C05459=1024.143,54.975,397.669,167.560,48.444,158.955
C05460=1024.137,54.725,397.687,167.557,48.448,158.956
C05461=1024.131,54.476,397.703,167.554,48.453,158.956
C05462=1024.125,54.227,397.719,167.551,48.457,158.956
C05463=1024.119,53.977,397.736,167.549,48.461,158.957
C05464=1024.113,53.728,397.752,167.547,48.465,158.957
C05465=1024.107,53.479,397.769,167.544,48.469,158.958
C05466=1024.102,53.230,397.786,167.542,48.473,158.958
C05467=1024.095,52.980,397.802,167.539,48.477,158.958
C05468=1024.089,52.730,397.818,167.536,48.481,158.959
C05469=1024.083,52.481,397.835,167.534,48.485,158.959
C05470=1024.077,52.232,397.852,167.531,48.489,158.960
C05471=1024.071,51.983,397.868,167.528,48.494,158.960
C05472=1024.066,51.733,397.885,167.527,48.497,158.961
C05473=1024.060,51.484,397.901,167.524,48.501,158.961
C05474=1024.054,51.234,397.917,167.521,48.505,158.961
C05475=1024.048,50.985,397.934,167.519,48.510,158.962
C05476=1024.041,50.735,397.950,167.516,48.513,158.962
C05477=1024.035,50.486,397.967,167.513,48.517,158.962
C05478=1024.030,50.237,397.984,167.510,48.521,158.963
C05479=1024.024,49.987,398.000,167.508,48.525,158.963
C05480=1024.018,49.738,398.017,167.506,48.529,158.964
C05481=1024.012,49.489,398.033,167.503,48.533,158.964
C05482=1024.006,49.239,398.049,167.500,48.537,158.964
C05483=1024.000,48.990,398.065,167.498,48.541,158.965
C05484=1023.995,48.740,398.082,167.495,48.546,158.965
C05485=1023.989,48.491,398.098,167.493,48.549,158.966
C05486=1023.983,48.242,398.115,167.491,48.553,158.966
C05487=1023.977,47.992,398.131,167.488,48.557,158.966
C05488=1023.971,47.743,398.147,167.485,48.561,158.967
C05489=1023.965,47.494,398.164,167.483,48.566,158.967
C05490=1023.959,47.245,398.180,167.480,48.570,158.968
C05491=1023.954,46.995,398.197,167.478,48.573,158.968
C05492=1023.948,46.746,398.214,167.475,48.577,158.968
C05493=1023.942,46.496,398.230,167.472,48.581,158.969
C05494=1023.935,46.246,398.246,167.470,48.585,158.969
C05495=1023.929,45.997,398.263,167.467,48.589,158.969
C05496=1023.923,45.748,398.279,167.464,48.593,158.970
C05497=1023.917,45.498,398.295,167.463,48.597,158.970
C05498=1023.912,45.249,398.312,167.460,48.601,158.971
C05499=1023.906,44.999,398.328,167.457,48.605,158.971
C05500=1023.901,44.751,398.344,167.454,48.609,158.971
C05501=1023.895,44.501,398.360,167.452,48.613,158.972
C05502=1023.889,44.252,398.377,167.449,48.617,158.972
C05503=1023.883,44.003,398.393,167.447,48.621,158.973
C05504=1023.876,43.717,398.411,167.444,48.625,158.973
C05505=1023.870,43.433,398.430,167.441,48.630,158.973
C05506=1023.863,43.148,398.449,167.439,48.634,158.974
C05507=1023.857,42.863,398.467,167.435,48.638,158.974
C05508=1023.851,42.614,398.484,167.432,48.642,158.974
C05509=1023.845,42.364,398.499,167.431,48.647,158.975
C05510=1023.839,42.115,398.516,167.428,48.651,158.975
C05511=1023.833,41.865,398.531,167.425,48.654,158.976
C05512=1023.827,41.616,398.547,167.422,48.658,158.976
C05513=1023.821,41.366,398.564,167.420,48.663,158.977
C05514=1023.815,41.117,398.580,167.417,48.667,158.977
C05515=1023.809,40.868,398.596,167.414,48.671,158.977
C05516=1023.804,40.618,398.612,167.412,48.675,158.978
C05517=1023.797,40.369,398.627,167.409,48.679,158.978
C05518=1023.791,40.119,398.644,167.407,48.683,158.978
C05519=1023.785,39.870,398.660,167.405,48.687,158.979
C05520=1023.779,39.620,398.675,167.402,48.691,158.979
C05521=1023.773,39.371,398.692,167.399,48.695,158.980
C05522=1023.767,39.121,398.708,167.397,48.699,158.980
C05523=1023.761,38.872,398.724,167.394,48.703,158.980
C05524=1023.756,38.623,398.739,167.391,48.707,158.981
C05525=1023.750,38.374,398.755,167.388,48.711,158.981
C05526=1023.744,38.124,398.771,167.387,48.715,158.982
C05527=1023.738,37.874,398.787,167.384,48.719,158.982
C05528=1023.732,37.625,398.803,167.381,48.723,158.982
C05529=1023.726,37.376,398.819,167.378,48.727,158.983
C05530=1023.720,37.126,398.834,167.376,48.731,158.983
C05531=1023.714,36.877,398.850,167.373,48.736,158.983
C05532=1023.708,36.627,398.867,167.370,48.740,158.984
C05533=1023.702,36.377,398.882,167.368,48.744,158.984
C05534=1023.696,36.129,398.898,167.365,48.747,158.984
C05535=1023.691,35.879,398.913,167.363,48.752,158.985
C05536=1023.684,35.630,398.929,167.361,48.756,158.985
C05537=1023.678,35.380,398.944,167.358,48.760,158.986
C05538=1023.672,35.131,398.961,167.356,48.764,158.986
C05539=1023.666,34.881,398.975,167.353,48.768,158.987
C05540=1023.660,34.632,398.992,167.350,48.772,158.987
C05541=1023.654,34.382,399.007,167.348,48.777,158.987
C05542=1023.648,34.133,399.023,167.345,48.781,158.988
C05543=1023.643,33.883,399.038,167.342,48.785,158.988
C05544=1023.636,33.634,399.054,167.339,48.789,158.988
C05545=1023.630,33.384,399.069,167.337,48.793,158.989
C05546=1023.624,33.135,399.085,167.334,48.797,158.989
C05547=1023.618,32.885,399.101,167.331,48.801,158.990
C05548=1023.612,32.636,399.117,167.329,48.805,158.990
C05549=1023.606,32.387,399.131,167.327,48.809,158.991
C05550=1023.600,32.138,399.148,167.324,48.813,158.991
C05551=1023.594,31.888,399.163,167.322,48.817,158.991
C05552=1023.588,31.639,399.179,167.319,48.821,158.992
C05553=1023.582,31.389,399.194,167.316,48.826,158.992
C05554=1023.576,31.141,399.210,167.314,48.830,158.992
C05555=1023.571,30.891,399.225,167.311,48.834,158.993
C05556=1023.564,30.641,399.240,167.308,48.837,158.993
C05557=1023.558,30.392,399.256,167.305,48.841,158.993
C05558=1023.553,30.142,399.272,167.303,48.846,158.994
C05559=1023.546,29.893,399.287,167.300,48.850,158.994
C05560=1023.541,29.643,399.303,167.298,48.854,158.995
C05561=1023.534,29.394,399.318,167.296,48.858,158.995
C05562=1023.528,29.144,399.334,167.293,48.861,158.995
C05563=1023.523,28.894,399.350,167.290,48.866,158.996
C05564=1023.517,28.645,399.364,167.288,48.870,158.996
C05565=1023.511,28.396,399.380,167.285,48.874,158.996
C05566=1023.505,28.146,399.395,167.282,48.878,158.997
C05567=1023.499,27.897,399.412,167.279,48.882,158.997
C05568=1023.492,27.612,399.428,167.277,48.887,158.998
C05569=1023.485,27.327,399.445,167.273,48.891,158.998
C05570=1023.479,27.043,399.463,167.271,48.896,158.999
C05571=1023.472,26.758,399.481,167.268,48.901,158.999
C05572=1023.466,26.508,399.496,167.265,48.905,158.999
C05573=1023.460,26.259,399.512,167.262,48.909,159.000
C05574=1023.453,26.009,399.527,167.259,48.913,159.000
C05575=1023.448,25.760,399.542,167.257,48.917,159.000
C05576=1023.442,25.510,399.557,167.255,48.921,159.001
C05577=1023.435,25.261,399.573,167.252,48.925,159.001
C05578=1023.430,25.011,399.588,167.250,48.929,159.002
C05579=1023.424,24.762,399.603,167.247,48.934,159.002
C05580=1023.417,24.513,399.618,167.244,48.938,159.002
C05581=1023.412,24.263,399.633,167.242,48.942,159.003
C05582=1023.406,24.014,399.648,167.239,48.945,159.003
C05583=1023.399,23.765,399.663,167.237,48.950,159.004
C05584=1023.394,23.515,399.679,167.234,48.954,159.004
C05585=1023.388,23.266,399.694,167.231,48.958,159.004
C05586=1023.381,23.016,399.709,167.228,48.962,159.005
C05587=1023.376,22.766,399.724,167.226,48.967,159.005
C05588=1023.369,22.517,399.739,167.223,48.971,159.005
C05589=1023.364,22.268,399.754,167.220,48.974,159.006
C05590=1023.358,22.018,399.769,167.218,48.978,159.006
C05591=1023.352,21.768,399.784,167.215,48.982,159.006
C05592=1023.346,21.520,399.799,167.212,48.987,159.007
C05593=1023.340,21.270,399.815,167.210,48.991,159.007
C05594=1023.334,21.020,399.830,167.207,48.995,159.008
C05595=1023.328,20.771,399.844,167.205,48.999,159.008
C05596=1023.322,20.521,399.860,167.202,49.003,159.008
C05597=1023.316,20.272,399.875,167.200,49.006,159.009
C05598=1023.310,20.023,399.890,167.197,49.011,159.009
C05599=1023.304,19.773,399.905,167.194,49.015,159.009
C05600=1023.299,19.524,399.920,167.192,49.019,159.010
C05601=1023.292,19.274,399.935,167.189,49.023,159.010
C05602=1023.286,19.024,399.950,167.186,49.027,159.010
C05603=1023.281,18.775,399.965,167.184,49.032,159.011
C05604=1023.274,18.525,399.980,167.181,49.036,159.011
C05605=1023.268,18.276,399.995,167.178,49.039,159.012
C05606=1023.262,18.027,400.009,167.175,49.043,159.012
C05607=1023.257,17.777,400.025,167.173,49.047,159.012
C05608=1023.251,17.528,400.039,167.170,49.052,159.013
C05609=1023.245,17.278,400.054,167.168,49.056,159.013
C05610=1023.238,17.028,400.068,167.165,49.060,159.013
C05611=1023.232,16.779,400.083,167.162,49.064,159.014
C05612=1023.226,16.529,400.098,167.160,49.069,159.014
C05613=1023.221,16.280,400.113,167.157,49.073,159.015
C05614=1023.215,16.030,400.128,167.154,49.077,159.015
C05615=1023.209,15.781,400.143,167.151,49.080,159.015
C05616=1023.203,15.532,400.158,167.149,49.084,159.015
C05617=1023.196,15.282,400.173,167.146,49.088,159.016
C05618=1023.191,15.032,400.187,167.144,49.093,159.016
C05619=1023.185,14.783,400.202,167.142,49.097,159.017
C05620=1023.179,14.534,400.217,167.139,49.101,159.017
C05621=1023.173,14.284,400.232,167.136,49.105,159.017
C05622=1023.167,14.035,400.246,167.134,49.109,159.018
C05623=1023.161,13.785,400.261,167.131,49.113,159.018
C05624=1023.156,13.535,400.276,167.128,49.117,159.018
C05625=1023.150,13.286,400.290,167.126,49.121,159.019
C05626=1023.142,13.036,400.305,167.123,49.125,159.019
C05627=1023.137,12.787,400.319,167.120,49.129,159.020
C05628=1023.131,12.537,400.334,167.118,49.134,159.020
C05629=1023.125,12.288,400.348,167.115,49.138,159.020
C05630=1023.119,12.038,400.362,167.112,49.142,159.021
C05631=1023.113,11.789,400.377,167.109,49.147,159.021
C05632=1023.106,11.506,400.393,167.106,49.151,159.021
C05633=1023.099,11.222,400.410,167.103,49.156,159.022
C05634=1023.092,10.939,400.426,167.100,49.160,159.022
C05635=1023.085,10.656,400.442,167.097,49.165,159.023
C05636=1023.079,10.406,400.457,167.094,49.169,159.023
C05637=1023.073,10.157,400.472,167.092,49.174,159.024
C05638=1023.067,9.907,400.486,167.089,49.178,159.024
C05639=1023.061,9.658,400.500,167.086,49.182,159.024
C05640=1023.055,9.408,400.515,167.083,49.186,159.024
C05641=1023.049,9.159,400.529,167.081,49.190,159.025
C05642=1023.043,8.909,400.544,167.078,49.194,159.025
C05643=1023.037,8.660,400.558,167.076,49.198,159.026
C05644=1023.030,8.410,400.572,167.073,49.202,159.026
C05645=1023.025,8.161,400.586,167.070,49.207,159.026
C05646=1023.018,7.911,400.601,167.068,49.211,159.027
C05647=1023.013,7.662,400.616,167.065,49.215,159.027
C05648=1023.007,7.412,400.630,167.062,49.219,159.027
C05649=1023.001,7.163,400.645,167.059,49.223,159.028
C05650=1022.995,6.913,400.659,167.057,49.228,159.028
C05651=1022.989,6.664,400.673,167.054,49.232,159.029
C05652=1022.984,6.414,400.687,167.052,49.236,159.029
C05653=1022.976,6.165,400.702,167.049,49.240,159.029
C05654=1022.971,5.915,400.715,167.046,49.244,159.030
C05655=1022.965,5.665,400.730,167.044,49.248,159.030
C05656=1022.959,5.416,400.744,167.041,49.252,159.030
C05657=1022.953,5.167,400.759,167.038,49.256,159.031
C05658=1022.947,4.917,400.773,167.035,49.260,159.031
C05659=1022.941,4.668,400.788,167.033,49.264,159.031
C05660=1022.935,4.417,400.802,167.030,49.268,159.032
C05661=1022.929,4.169,400.816,167.027,49.272,159.032
C05662=1022.923,3.919,400.830,167.025,49.277,159.032
C05663=1022.917,3.669,400.844,167.022,49.281,159.033
C05664=1022.911,3.420,400.859,167.019,49.285,159.033
C05665=1022.905,3.170,400.873,167.017,49.289,159.033
C05666=1022.900,2.921,400.887,167.014,49.293,159.034
C05667=1022.894,2.671,400.901,167.011,49.297,159.034
C05668=1022.887,2.421,400.915,167.008,49.301,159.034
C05669=1022.882,2.172,400.929,167.006,49.305,159.035
C05670=1022.876,1.923,400.943,167.003,49.309,159.035
C05671=1022.870,1.673,400.958,167.001,49.313,159.035
C05672=1022.864,1.423,400.972,166.998,49.317,159.036
C05673=1022.859,1.174,400.986,166.995,49.321,159.036
C05674=1022.852,0.924,401.001,166.992,49.325,159.036
C05675=1022.846,0.675,401.014,166.990,49.329,159.037
C05676=1022.841,0.425,401.028,166.987,49.333,159.037
C05677=1022.834,0.176,401.043,166.984,49.337,159.037
C05678=1022.829,-0.074,401.057,166.981,49.341,159.038
C05679=1022.823,-0.324,401.071,166.979,49.345,159.038
C05680=1022.818,-0.572,401.085,166.976,49.349,159.038
C05681=1022.811,-0.823,401.100,166.973,49.353,159.039
C05682=1022.805,-1.072,401.113,166.970,49.357,159.039
C05683=1022.799,-1.321,401.127,166.968,49.361,159.039
C05684=1022.793,-1.571,401.142,166.965,49.365,159.040
C05685=1022.788,-1.821,401.155,166.962,49.369,159.040
C05686=1022.782,-2.070,401.170,166.960,49.373,159.040
C05687=1022.777,-2.319,401.184,166.957,49.377,159.041
C05688=1022.771,-2.570,401.198,166.954,49.381,159.041
C05689=1022.764,-2.819,401.211,166.951,49.385,159.041
C05690=1022.759,-3.068,401.226,166.949,49.389,159.042
C05691=1022.753,-3.317,401.240,166.946,49.393,159.042
C05692=1022.747,-3.568,401.254,166.943,49.397,159.042
C05693=1022.742,-3.817,401.268,166.940,49.401,159.042
C05694=1022.736,-4.067,401.282,166.938,49.405,159.043
C05695=1022.730,-4.315,401.296,166.935,49.410,159.043
C05696=1022.722,-4.598,401.311,166.932,49.414,159.043
C05697=1022.715,-4.879,401.327,166.928,49.419,159.044
C05698=1022.709,-5.161,401.342,166.926,49.424,159.044
C05699=1022.702,-5.442,401.358,166.922,49.429,159.045
C05700=1022.696,-5.691,401.372,166.920,49.433,159.045
C05701=1022.690,-5.941,401.385,166.917,49.437,159.045
C05702=1022.685,-6.190,401.399,166.914,49.441,159.046
C05703=1022.678,-6.440,401.412,166.911,49.445,159.046
C05704=1022.672,-6.690,401.426,166.909,49.449,159.047
C05705=1022.666,-6.939,401.439,166.906,49.453,159.047
C05706=1022.661,-7.189,401.453,166.904,49.457,159.047
C05707=1022.655,-7.438,401.467,166.900,49.462,159.047
C05708=1022.648,-7.688,401.481,166.897,49.466,159.048
C05709=1022.642,-7.937,401.494,166.894,49.470,159.048
C05710=1022.637,-8.187,401.508,166.892,49.474,159.048
C05711=1022.631,-8.436,401.521,166.889,49.478,159.049
C05712=1022.625,-8.686,401.535,166.887,49.482,159.049
C05713=1022.619,-8.935,401.548,166.884,49.486,159.049
C05714=1022.613,-9.185,401.563,166.881,49.490,159.050
C05715=1022.607,-9.435,401.576,166.878,49.495,159.050
C05716=1022.601,-9.685,401.589,166.876,49.499,159.050
C05717=1022.595,-9.934,401.602,166.873,49.503,159.051
C05718=1022.590,-10.184,401.616,166.871,49.507,159.051
C05719=1022.583,-10.433,401.629,166.867,49.512,159.051
C05720=1022.577,-10.682,401.643,166.864,49.516,159.052
C05721=1022.571,-10.933,401.657,166.861,49.520,159.052
C05722=1022.565,-11.182,401.670,166.859,49.524,159.052
C05723=1022.559,-11.431,401.684,166.856,49.528,159.053
C05724=1022.553,-11.681,401.697,166.853,49.532,159.053
C05725=1022.548,-11.930,401.711,166.851,49.536,159.053
C05726=1022.542,-12.180,401.724,166.848,49.540,159.054
C05727=1022.536,-12.430,401.738,166.845,49.544,159.054
C05728=1022.530,-12.679,401.751,166.842,49.548,159.054
C05729=1022.525,-12.928,401.765,166.840,49.552,159.054
C05730=1022.518,-13.178,401.778,166.837,49.556,159.055
C05731=1022.512,-13.428,401.792,166.835,49.560,159.055
C05732=1022.507,-13.678,401.805,166.832,49.564,159.056
C05733=1022.501,-13.928,401.819,166.828,49.569,159.056
C05734=1022.495,-14.177,401.832,166.825,49.573,159.056
C05735=1022.489,-14.426,401.845,166.823,49.577,159.056
C05736=1022.483,-14.676,401.859,166.820,49.581,159.057
C05737=1022.477,-14.925,401.872,166.817,49.585,159.057
C05738=1022.472,-15.175,401.885,166.814,49.589,159.057
C05739=1022.466,-15.424,401.899,166.812,49.593,159.058
C05740=1022.460,-15.674,401.913,166.809,49.597,159.058
C05741=1022.454,-15.924,401.925,166.806,49.601,159.058
C05742=1022.448,-16.173,401.938,166.804,49.605,159.059
C05743=1022.442,-16.422,401.952,166.801,49.609,159.059
C05744=1022.437,-16.673,401.965,166.797,49.613,159.059
C05745=1022.430,-16.922,401.978,166.795,49.618,159.060
C05746=1022.424,-17.172,401.991,166.792,49.622,159.060
C05747=1022.418,-17.421,402.004,166.789,49.626,159.060
C05748=1022.412,-17.670,402.017,166.787,49.630,159.061
C05749=1022.407,-17.920,402.030,166.784,49.634,159.061
C05750=1022.401,-18.170,402.044,166.781,49.638,159.061
C05751=1022.395,-18.420,402.056,166.777,49.642,159.061
C05752=1022.389,-18.669,402.069,166.775,49.647,159.062
C05753=1022.383,-18.919,402.082,166.772,49.651,159.062
C05754=1022.377,-19.168,402.096,166.770,49.655,159.062
C05755=1022.371,-19.417,402.109,166.767,49.659,159.063
C05756=1022.365,-19.667,402.122,166.764,49.663,159.063
C05757=1022.359,-19.917,402.135,166.762,49.667,159.063
C05758=1022.353,-20.167,402.148,166.758,49.671,159.064
C05759=1022.347,-20.416,402.161,166.755,49.675,159.064
C05760=1022.340,-20.696,402.176,166.753,49.680,159.064
C05761=1022.334,-20.976,402.191,166.749,49.685,159.065
C05762=1022.327,-21.255,402.205,166.746,49.690,159.065
C05763=1022.320,-21.535,402.220,166.743,49.694,159.065
C05764=1022.314,-21.785,402.232,166.740,49.698,159.066
C05765=1022.309,-22.035,402.245,166.738,49.702,159.066
C05766=1022.302,-22.284,402.258,166.734,49.707,159.066
C05767=1022.297,-22.533,402.270,166.731,49.711,159.067
C05768=1022.292,-22.783,402.284,166.729,49.715,159.067
C05769=1022.286,-23.033,402.297,166.726,49.719,159.067
C05770=1022.279,-23.282,402.310,166.723,49.723,159.067
C05771=1022.274,-23.532,402.323,166.720,49.727,159.068
C05772=1022.267,-23.781,402.336,166.718,49.731,159.068
C05773=1022.261,-24.031,402.348,166.715,49.735,159.068
C05774=1022.256,-24.281,402.362,166.711,49.739,159.069
C05775=1022.250,-24.530,402.375,166.709,49.743,159.069
C05776=1022.244,-24.780,402.387,166.706,49.747,159.069
C05777=1022.238,-25.029,402.400,166.703,49.751,159.069
C05778=1022.233,-25.279,402.413,166.700,49.755,159.070
C05779=1022.227,-25.529,402.425,166.698,49.759,159.070
C05780=1022.221,-25.778,402.439,166.695,49.763,159.070
C05781=1022.215,-26.028,402.452,166.692,49.767,159.071
C05782=1022.209,-26.278,402.464,166.689,49.772,159.071
C05783=1022.204,-26.527,402.477,166.686,49.776,159.071
C05784=1022.198,-26.776,402.490,166.683,49.780,159.072
C05785=1022.192,-27.026,402.502,166.681,49.784,159.072
C05786=1022.186,-27.276,402.516,166.678,49.788,159.072
C05787=1022.181,-27.526,402.529,166.675,49.792,159.072
C05788=1022.175,-27.776,402.541,166.672,49.796,159.073
C05789=1022.168,-28.025,402.553,166.669,49.800,159.073
C05790=1022.163,-28.274,402.565,166.666,49.804,159.073
C05791=1022.156,-28.524,402.579,166.664,49.809,159.074
C05792=1022.151,-28.774,402.591,166.661,49.813,159.074
C05793=1022.145,-29.023,402.604,166.658,49.817,159.074
C05794=1022.139,-29.273,402.616,166.654,49.822,159.074
C05795=1022.133,-29.523,402.629,166.652,49.826,159.075
C05796=1022.128,-29.772,402.641,166.649,49.830,159.075
C05797=1022.122,-30.022,402.654,166.646,49.834,159.075
C05798=1022.115,-30.271,402.666,166.644,49.838,159.076
C05799=1022.109,-30.521,402.679,166.641,49.842,159.076
C05800=1022.103,-30.770,402.691,166.638,49.847,159.076
C05801=1022.098,-31.020,402.704,166.635,49.851,159.077
C05802=1022.092,-31.270,402.716,166.632,49.855,159.077
C05803=1022.086,-31.520,402.729,166.629,49.859,159.077
C05804=1022.080,-31.770,402.741,166.627,49.863,159.078
C05805=1022.075,-32.019,402.754,166.623,49.867,159.078
C05806=1022.068,-32.269,402.765,166.620,49.871,159.078
C05807=1022.062,-32.518,402.778,166.618,49.875,159.078
C05808=1022.057,-32.768,402.790,166.615,49.880,159.079
C05809=1022.051,-33.018,402.803,166.612,49.884,159.079
C05810=1022.045,-33.267,402.816,166.608,49.888,159.079
C05811=1022.039,-33.517,402.829,166.606,49.892,159.079
C05812=1022.033,-33.766,402.841,166.603,49.896,159.080
C05813=1022.027,-34.015,402.853,166.600,49.900,159.080
C05814=1022.021,-34.265,402.865,166.598,49.904,159.080
C05815=1022.015,-34.514,402.877,166.594,49.908,159.081
C05816=1022.010,-34.764,402.890,166.591,49.913,159.081
C05817=1022.004,-35.014,402.903,166.589,49.917,159.081
C05818=1021.998,-35.263,402.915,166.586,49.921,159.081
C05819=1021.992,-35.513,402.927,166.583,49.925,159.082
C05820=1021.986,-35.764,402.939,166.580,49.929,159.082
C05821=1021.981,-36.013,402.951,166.577,49.933,159.082
C05822=1021.975,-36.263,402.963,166.574,49.937,159.083
C05823=1021.969,-36.512,402.976,166.571,49.941,159.083
C05824=1021.962,-36.791,402.989,166.568,49.946,159.083
C05825=1021.956,-37.070,403.004,166.565,49.950,159.084
C05826=1021.949,-37.349,403.017,166.562,49.955,159.084
C05827=1021.943,-37.627,403.031,166.558,49.960,159.084
C05828=1021.938,-37.878,403.043,166.555,49.964,159.084
C05829=1021.932,-38.127,403.055,166.553,49.968,159.085
C05830=1021.926,-38.376,403.067,166.550,49.972,159.085
C05831=1021.920,-38.626,403.080,166.547,49.976,159.085
C05832=1021.915,-38.876,403.092,166.545,49.980,159.086
C05833=1021.909,-39.125,403.105,166.541,49.984,159.086
C05834=1021.903,-39.375,403.117,166.538,49.988,159.086
C05835=1021.897,-39.625,403.128,166.536,49.993,159.086
C05836=1021.891,-39.875,403.141,166.533,49.997,159.087
C05837=1021.885,-40.124,403.152,166.529,50.001,159.087
C05838=1021.880,-40.374,403.164,166.526,50.005,159.087
C05839=1021.873,-40.624,403.176,166.524,50.009,159.087
C05840=1021.868,-40.873,403.188,166.521,50.013,159.088
C05841=1021.862,-41.123,403.201,166.517,50.018,159.088
C05842=1021.856,-41.372,403.212,166.515,50.022,159.088
C05843=1021.850,-41.622,403.224,166.512,50.026,159.089
C05844=1021.844,-41.871,403.236,166.510,50.030,159.089
C05845=1021.838,-42.121,403.247,166.506,50.035,159.089
C05846=1021.832,-42.371,403.260,166.503,50.039,159.089
C05847=1021.826,-42.620,403.272,166.501,50.043,159.090
C05848=1021.821,-42.871,403.283,166.498,50.047,159.090
C05849=1021.815,-43.120,403.295,166.494,50.051,159.090
C05850=1021.809,-43.369,403.308,166.491,50.055,159.091
C05851=1021.803,-43.619,403.319,166.489,50.059,159.091
C05852=1021.797,-43.869,403.331,166.486,50.064,159.091
C05853=1021.792,-44.119,403.343,166.483,50.068,159.091
C05854=1021.786,-44.368,403.354,166.480,50.072,159.092
C05855=1021.780,-44.617,403.367,166.477,50.076,159.092
C05856=1021.774,-44.868,403.378,166.474,50.080,159.092
C05857=1021.769,-45.117,403.390,166.472,50.084,159.092
C05858=1021.762,-45.367,403.401,166.468,50.089,159.093
C05859=1021.757,-45.616,403.414,166.465,50.093,159.093
C05860=1021.751,-45.866,403.425,166.462,50.097,159.093
C05861=1021.745,-46.115,403.437,166.460,50.101,159.094
C05862=1021.740,-46.366,403.449,166.456,50.105,159.094
C05863=1021.734,-46.615,403.460,166.453,50.109,159.094
C05864=1021.728,-46.865,403.473,166.451,50.113,159.094
C05865=1021.722,-47.114,403.484,166.448,50.117,159.095
C05866=1021.717,-47.363,403.496,166.445,50.121,159.095
C05867=1021.710,-47.614,403.507,166.442,50.126,159.095
C05868=1021.705,-47.863,403.519,166.439,50.130,159.095
C05869=1021.699,-48.113,403.531,166.436,50.134,159.096
C05870=1021.693,-48.362,403.543,166.434,50.138,159.096
C05871=1021.688,-48.613,403.555,166.430,50.142,159.096
C05872=1021.682,-48.862,403.566,166.427,50.147,159.096
C05873=1021.677,-49.111,403.578,166.424,50.150,159.097
C05874=1021.670,-49.362,403.589,166.421,50.154,159.097
C05875=1021.665,-49.611,403.601,166.419,50.158,159.097
C05876=1021.659,-49.861,403.612,166.415,50.162,159.097
C05877=1021.653,-50.110,403.625,166.412,50.167,159.098
C05878=1021.648,-50.360,403.636,166.410,50.171,159.098
C05879=1021.642,-50.610,403.647,166.407,50.175,159.098
C05880=1021.636,-50.859,403.659,166.403,50.179,159.098
C05881=1021.631,-51.109,403.670,166.401,50.183,159.099
C05882=1021.625,-51.359,403.682,166.398,50.187,159.099
C05883=1021.619,-51.608,403.693,166.394,50.192,159.099
C05884=1021.612,-51.858,403.705,166.392,50.196,159.099
C05885=1021.607,-52.107,403.715,166.389,50.201,159.100
C05886=1021.602,-52.357,403.727,166.385,50.205,159.100
C05887=1021.595,-52.607,403.738,166.383,50.209,159.100
C05888=1021.589,-52.855,403.749,166.380,50.213,159.101
C05889=1021.583,-53.103,403.761,166.376,50.217,159.101
C05890=1021.578,-53.350,403.771,166.374,50.222,159.101
C05891=1021.572,-53.597,403.783,166.371,50.226,159.101
C05892=1021.566,-53.845,403.794,166.368,50.231,159.102
C05893=1021.560,-54.093,403.805,166.365,50.235,159.102
C05894=1021.554,-54.341,403.815,166.362,50.239,159.102
C05895=1021.548,-54.589,403.827,166.360,50.243,159.103
C05896=1021.543,-54.838,403.838,166.356,50.247,159.103
C05897=1021.537,-55.088,403.849,166.353,50.251,159.103
C05898=1021.531,-55.338,403.860,166.351,50.256,159.103
C05899=1021.525,-55.587,403.871,166.347,50.260,159.103
C05900=1021.520,-55.837,403.883,166.344,50.264,159.104
C05901=1021.514,-56.087,403.894,166.342,50.268,159.104
C05902=1021.508,-56.337,403.905,166.338,50.273,159.104
C05903=1021.502,-56.586,403.916,166.335,50.277,159.105
C05904=1021.496,-56.835,403.927,166.333,50.281,159.105
C05905=1021.490,-57.085,403.938,166.329,50.286,159.105
C05906=1021.484,-57.335,403.949,166.326,50.290,159.105
C05907=1021.478,-57.584,403.960,166.324,50.294,159.106
C05908=1021.472,-57.868,403.973,166.320,50.299,159.106
C05909=1021.465,-58.151,403.985,166.317,50.304,159.106
C05910=1021.459,-58.434,403.998,166.313,50.309,159.107
C05911=1021.452,-58.717,404.010,166.310,50.313,159.107
C05912=1021.447,-58.968,404.022,166.307,50.317,159.107
C05913=1021.441,-59.217,404.033,166.303,50.322,159.107
C05914=1021.435,-59.467,404.044,166.301,50.326,159.108
C05915=1021.429,-59.716,404.055,166.298,50.330,159.108
C05916=1021.424,-59.966,404.065,166.294,50.334,159.108
C05917=1021.417,-60.216,404.077,166.292,50.338,159.108
C05918=1021.411,-60.465,404.088,166.289,50.342,159.109
C05919=1021.406,-60.715,404.098,166.285,50.347,159.109
C05920=1021.401,-60.964,404.110,166.283,50.352,159.109
C05921=1021.395,-61.214,404.121,166.280,50.356,159.110
C05922=1021.389,-61.463,404.132,166.277,50.359,159.110
C05923=1021.383,-61.714,404.142,166.273,50.363,159.110
C05924=1021.377,-61.964,404.153,166.271,50.368,159.110
C05925=1021.372,-62.213,404.164,166.268,50.372,159.110
C05926=1021.366,-62.463,404.175,166.264,50.376,159.111
C05927=1021.360,-62.712,404.186,166.262,50.380,159.111
C05928=1021.355,-62.962,404.197,166.259,50.384,159.111
C05929=1021.350,-63.212,404.208,166.255,50.389,159.111
C05930=1021.343,-63.462,404.219,166.253,50.393,159.112
C05931=1021.338,-63.712,404.229,166.250,50.397,159.112
C05932=1021.332,-63.961,404.240,166.246,50.401,159.112
C05933=1021.326,-64.211,404.251,166.244,50.405,159.112
C05934=1021.321,-64.460,404.262,166.241,50.410,159.113
C05935=1021.315,-64.710,404.273,166.238,50.414,159.113
C05936=1021.309,-64.959,404.284,166.235,50.418,159.113
C05937=1021.304,-65.209,404.294,166.232,50.422,159.113
C05938=1021.298,-65.459,404.305,166.229,50.426,159.114
C05939=1021.293,-65.709,404.316,166.226,50.431,159.114
C05940=1021.287,-65.958,404.327,166.223,50.435,159.114
C05941=1021.282,-66.208,404.337,166.220,50.438,159.114
C05942=1021.276,-66.458,404.348,166.217,50.442,159.114
C05943=1021.270,-66.708,404.360,166.213,50.447,159.115
C05944=1021.264,-66.957,404.370,166.211,50.451,159.115
C05945=1021.258,-67.208,404.381,166.208,50.455,159.115
C05946=1021.253,-67.457,404.391,166.204,50.459,159.115
C05947=1021.247,-67.707,404.402,166.202,50.463,159.116
C05948=1021.241,-67.956,404.413,166.199,50.468,159.116
C05949=1021.236,-68.206,404.423,166.196,50.472,159.116
C05950=1021.230,-68.456,404.434,166.192,50.475,159.116
C05951=1021.225,-68.705,404.446,166.190,50.480,159.116
C05952=1021.219,-68.986,404.457,166.186,50.485,159.117
C05953=1021.213,-69.266,404.469,166.184,50.489,159.117
C05954=1021.207,-69.547,404.481,166.180,50.493,159.117
C05955=1021.201,-69.826,404.493,166.177,50.498,159.117
C05956=1021.195,-70.076,404.504,166.174,50.502,159.118
C05957=1021.189,-70.326,404.514,166.170,50.506,159.118
C05958=1021.184,-70.576,404.525,166.167,50.510,159.118
C05959=1021.178,-70.825,404.536,166.165,50.514,159.118
C05960=1021.172,-71.075,404.546,166.162,50.519,159.119
C05961=1021.167,-71.325,404.557,166.158,50.522,159.119
C05962=1021.161,-71.575,404.567,166.155,50.526,159.119
C05963=1021.156,-71.824,404.578,166.153,50.530,159.119
C05964=1021.150,-72.074,404.589,166.150,50.535,159.119
C05965=1021.144,-72.324,404.599,166.146,50.539,159.120
C05966=1021.139,-72.573,404.610,166.143,50.542,159.120
C05967=1021.133,-72.823,404.620,166.140,50.547,159.120
C05968=1021.129,-73.073,404.631,166.138,50.551,159.120
C05969=1021.123,-73.323,404.641,166.134,50.555,159.120
C05970=1021.118,-73.572,404.652,166.131,50.559,159.121
C05971=1021.112,-73.822,404.662,166.128,50.563,159.121
C05972=1021.106,-74.072,404.673,166.126,50.567,159.121
C05973=1021.101,-74.322,404.683,166.122,50.571,159.121
C05974=1021.095,-74.571,404.694,166.119,50.575,159.121
C05975=1021.090,-74.821,404.704,166.117,50.579,159.122
C05976=1021.083,-75.071,404.715,166.113,50.584,159.122
C05977=1021.079,-75.320,404.724,166.110,50.588,159.122
C05978=1021.073,-75.570,404.735,166.108,50.592,159.122
C05979=1021.067,-75.820,404.746,166.104,50.597,159.123
C05980=1021.061,-76.069,404.755,166.101,50.601,159.123
C05981=1021.056,-76.320,404.765,166.098,50.604,159.123
C05982=1021.050,-76.569,404.776,166.095,50.609,159.123
C05983=1021.045,-76.819,404.786,166.092,50.613,159.123
C05984=1021.039,-77.068,404.795,166.089,50.617,159.124
C05985=1021.033,-77.318,404.806,166.086,50.621,159.124
C05986=1021.028,-77.568,404.817,166.083,50.625,159.124
C05987=1021.022,-77.818,404.827,166.080,50.629,159.124
C05988=1021.016,-78.068,404.836,166.077,50.634,159.124
C05989=1021.011,-78.317,404.847,166.074,50.638,159.125
C05990=1021.006,-78.567,404.857,166.071,50.642,159.125
C05991=1021.000,-78.817,404.867,166.068,50.647,159.125
C05992=1020.994,-79.067,404.877,166.065,50.651,159.125
C05993=1020.988,-79.316,404.888,166.062,50.654,159.126
C05994=1020.983,-79.565,404.897,166.058,50.659,159.126
C05995=1020.978,-79.816,404.907,166.056,50.663,159.126
C05996=1020.972,-80.065,404.917,166.053,50.667,159.126
C05997=1020.966,-80.315,404.927,166.049,50.671,159.126
C05998=1020.962,-80.565,404.937,166.047,50.675,159.127
C05999=1020.955,-80.814,404.947,166.043,50.680,159.127
C06000=1020.950,-81.064,404.957,166.040,50.684,159.127
C06001=1020.944,-81.314,404.967,166.038,50.688,159.127
C06002=1020.939,-81.563,404.977,166.034,50.693,159.128
C06003=1020.933,-81.813,404.986,166.031,50.697,159.128
C06004=1020.927,-82.063,404.997,166.028,50.702,159.128
C06005=1020.921,-82.313,405.006,166.025,50.706,159.128
C06006=1020.915,-82.562,405.015,166.023,50.710,159.129
C06007=1020.910,-82.812,405.025,166.019,50.715,159.129
C06008=1020.904,-83.062,405.035,166.016,50.719,159.129
C06009=1020.898,-83.312,405.045,166.013,50.723,159.129
C06010=1020.893,-83.561,405.054,166.010,50.727,159.130
C06011=1020.887,-83.811,405.065,166.007,50.732,159.130
C06012=1020.881,-84.061,405.074,166.004,50.736,159.130
C06013=1020.876,-84.311,405.084,166.001,50.740,159.130
C06014=1020.870,-84.560,405.094,165.997,50.745,159.130
C06015=1020.865,-84.811,405.104,165.995,50.749,159.131
C06016=1020.859,-85.093,405.114,165.991,50.753,159.131
C06017=1020.852,-85.375,405.125,165.988,50.758,159.131
C06018=1020.846,-85.657,405.137,165.984,50.763,159.131
C06019=1020.840,-85.940,405.147,165.981,50.768,159.132
C06020=1020.834,-86.189,405.156,165.978,50.772,159.132
C06021=1020.829,-86.439,405.167,165.974,50.777,159.132
C06022=1020.822,-86.689,405.176,165.972,50.781,159.132
C06023=1020.818,-86.939,405.186,165.969,50.785,159.133
C06024=1020.811,-87.188,405.195,165.965,50.789,159.133
C06025=1020.806,-87.439,405.204,165.963,50.794,159.133
C06026=1020.801,-87.688,405.214,165.959,50.798,159.133
C06027=1020.795,-87.938,405.224,165.956,50.802,159.133
C06028=1020.790,-88.187,405.233,165.953,50.806,159.133
C06029=1020.784,-88.437,405.243,165.950,50.810,159.134
C06030=1020.778,-88.687,405.253,165.947,50.814,159.134
C06031=1020.773,-88.936,405.262,165.944,50.818,159.134
C06032=1020.767,-89.187,405.272,165.941,50.823,159.134
C06033=1020.762,-89.436,405.281,165.938,50.827,159.135
C06034=1020.756,-89.686,405.291,165.935,50.831,159.135
C06035=1020.751,-89.935,405.300,165.932,50.836,159.135
C06036=1020.745,-90.185,405.310,165.929,50.840,159.135
C06037=1020.740,-90.435,405.319,165.925,50.844,159.135
C06038=1020.734,-90.685,405.329,165.923,50.848,159.136
C06039=1020.729,-90.934,405.338,165.920,50.852,159.136
C06040=1020.723,-91.184,405.348,165.916,50.856,159.136
C06041=1020.718,-91.434,405.357,165.913,50.860,159.136
C06042=1020.712,-91.684,405.367,165.911,50.865,159.136
C06043=1020.707,-91.933,405.376,165.907,50.869,159.137
C06044=1020.702,-92.184,405.385,165.904,50.873,159.137
C06045=1020.696,-92.433,405.394,165.902,50.877,159.137
C06046=1020.691,-92.683,405.405,165.898,50.882,159.137
C06047=1020.685,-92.932,405.414,165.895,50.886,159.138
C06048=1020.680,-93.183,405.423,165.892,50.889,159.138
C06049=1020.674,-93.432,405.432,165.889,50.894,159.138
C06050=1020.669,-93.682,405.443,165.886,50.898,159.138
C06051=1020.664,-93.932,405.451,165.883,50.902,159.138
C06052=1020.657,-94.182,405.461,165.880,50.907,159.138
C06053=1020.653,-94.431,405.470,165.877,50.911,159.139
C06054=1020.647,-94.681,405.479,165.874,50.914,159.139
C06055=1020.642,-94.931,405.489,165.870,50.919,159.139
C06056=1020.637,-95.181,405.498,165.868,50.923,159.139
C06057=1020.631,-95.431,405.508,165.865,50.927,159.139
C06058=1020.626,-95.680,405.517,165.861,50.932,159.140
C06059=1020.620,-95.930,405.526,165.858,50.935,159.140
C06060=1020.615,-96.180,405.536,165.856,50.939,159.140
C06061=1020.609,-96.430,405.544,165.852,50.944,159.140
C06062=1020.604,-96.679,405.554,165.849,50.948,159.140
C06063=1020.599,-96.929,405.563,165.847,50.952,159.141
C06064=1020.593,-97.179,405.572,165.843,50.956,159.140
C06065=1020.588,-97.428,405.582,165.840,50.960,159.141
C06066=1020.582,-97.679,405.591,165.838,50.964,159.141
C06067=1020.577,-97.928,405.601,165.834,50.969,159.141
C06068=1020.572,-98.178,405.609,165.831,50.973,159.141
C06069=1020.566,-98.428,405.618,165.829,50.977,159.142
C06070=1020.561,-98.677,405.627,165.825,50.981,159.142
C06071=1020.555,-98.927,405.636,165.822,50.986,159.142
C06072=1020.549,-99.177,405.645,165.819,50.990,159.142
C06073=1020.545,-99.427,405.654,165.816,50.994,159.142
C06074=1020.539,-99.677,405.663,165.813,50.998,159.143
C06075=1020.533,-99.926,405.672,165.810,51.003,159.143
C06076=1020.528,-100.176,405.681,165.807,51.007,159.143
C06077=1020.523,-100.426,405.689,165.803,51.011,159.143
C06078=1020.516,-100.676,405.699,165.800,51.015,159.143
C06079=1020.511,-100.925,405.708,165.798,51.019,159.144
C06080=1020.505,-101.210,405.718,165.794,51.024,159.144
C06081=1020.499,-101.495,405.728,165.791,51.029,159.144
C06082=1020.493,-101.779,405.738,165.787,51.034,159.144
C06083=1020.486,-102.063,405.748,165.784,51.039,159.145
C06084=1020.482,-102.313,405.757,165.780,51.043,159.145
C06085=1020.476,-102.563,405.766,165.777,51.047,159.145
C06086=1020.470,-102.814,405.775,165.775,51.051,159.145
C06087=1020.465,-103.063,405.784,165.771,51.056,159.145
C06088=1020.460,-103.312,405.793,165.768,51.060,159.146
C06089=1020.454,-103.562,405.801,165.765,51.065,159.146
C06090=1020.448,-103.812,405.810,165.762,51.069,159.146
C06091=1020.443,-104.062,405.819,165.759,51.072,159.146
C06092=1020.438,-104.312,405.828,165.756,51.077,159.146
C06093=1020.433,-104.561,405.837,165.753,51.081,159.146
C06094=1020.427,-104.812,405.845,165.750,51.085,159.147
C06095=1020.422,-105.061,405.854,165.747,51.089,159.147
C06096=1020.416,-105.311,405.863,165.744,51.094,159.147
C06097=1020.411,-105.560,405.872,165.741,51.098,159.147
C06098=1020.406,-105.810,405.880,165.738,51.102,159.147
C06099=1020.400,-106.060,405.889,165.735,51.106,159.148
C06100=1020.395,-106.310,405.897,165.731,51.110,159.148
C06101=1020.389,-106.560,405.906,165.728,51.114,159.148
C06102=1020.384,-106.810,405.914,165.726,51.119,159.148
C06103=1020.379,-107.059,405.923,165.722,51.123,159.148
C06104=1020.373,-107.309,405.932,165.719,51.127,159.149
C06105=1020.367,-107.559,405.941,165.717,51.132,159.149
C06106=1020.363,-107.809,405.950,165.713,51.136,159.149
C06107=1020.357,-108.058,405.958,165.710,51.140,159.149
C06108=1020.352,-108.308,405.966,165.707,51.145,159.149
C06109=1020.346,-108.558,405.975,165.704,51.149,159.150
C06110=1020.341,-108.808,405.984,165.701,51.152,159.150
C06111=1020.335,-109.058,405.992,165.697,51.157,159.150
C06112=1020.330,-109.307,406.001,165.695,51.161,159.150
C06113=1020.325,-109.557,406.009,165.691,51.166,159.150
C06114=1020.319,-109.807,406.018,165.689,51.170,159.150
C06115=1020.314,-110.057,406.026,165.686,51.174,159.151
C06116=1020.309,-110.306,406.035,165.682,51.178,159.151
C06117=1020.304,-110.557,406.042,165.680,51.183,159.151
C06118=1020.299,-110.806,406.051,165.677,51.187,159.151
C06119=1020.292,-111.056,406.059,165.673,51.191,159.151
C06120=1020.287,-111.306,406.068,165.671,51.196,159.152
C06121=1020.282,-111.556,406.076,165.667,51.200,159.152
C06122=1020.276,-111.806,406.085,165.664,51.204,159.152
C06123=1020.271,-112.055,406.093,165.661,51.208,159.152
C06124=1020.266,-112.305,406.102,165.658,51.212,159.152
C06125=1020.261,-112.555,406.110,165.655,51.216,159.153
C06126=1020.255,-112.804,406.119,165.653,51.221,159.153
C06127=1020.250,-113.055,406.126,165.649,51.225,159.153
C06128=1020.245,-113.305,406.135,165.646,51.229,159.153
C06129=1020.239,-113.554,406.143,165.643,51.234,159.153
C06130=1020.234,-113.804,406.151,165.640,51.238,159.154
C06131=1020.229,-114.053,406.160,165.637,51.242,159.154
C06132=1020.223,-114.303,406.168,165.633,51.246,159.154
C06133=1020.218,-114.553,406.176,165.631,51.250,159.154
C06134=1020.213,-114.803,406.184,165.628,51.254,159.154
C06135=1020.208,-115.053,406.193,165.624,51.259,159.154
C06136=1020.202,-115.302,406.201,165.622,51.263,159.155
C06137=1020.197,-115.553,406.209,165.618,51.268,159.155
C06138=1020.192,-115.802,406.217,165.615,51.272,159.155
C06139=1020.186,-116.052,406.226,165.613,51.276,159.155
C06140=1020.180,-116.301,406.233,165.609,51.281,159.155
C06141=1020.175,-116.552,406.241,165.607,51.285,159.156
C06142=1020.170,-116.801,406.250,165.604,51.289,159.156
C06143=1020.165,-117.051,406.258,165.600,51.293,159.156
C06144=1020.159,-117.335,406.267,165.597,51.298,159.156
C06145=1020.152,-117.620,406.276,165.593,51.303,159.156
C06146=1020.146,-117.904,406.285,165.590,51.308,159.157
C06147=1020.140,-118.189,406.295,165.586,51.312,159.157
C06148=1020.135,-118.439,406.303,165.583,51.316,159.157
///RCONF 1,0,0,0,1,0,0,0,0,0,0,0,0,0,0,0,0,0,0,0,0,0,0,0
C06149=1020.130,-118.688,406.310,165.581,51.321,159.157
C06150=1020.125,-118.938,406.318,165.577,51.325,159.157
C06151=1020.120,-119.188,406.327,165.575,51.329,159.158
C06152=1020.114,-119.437,406.334,165.571,51.334,159.158
C06153=1020.109,-119.688,406.342,165.568,51.338,159.158
C06154=1020.103,-119.937,406.351,165.566,51.342,159.158
C06155=1020.098,-120.188,406.358,165.562,51.347,159.158
C06156=1020.092,-120.437,406.366,165.559,51.350,159.158
C06157=1020.088,-120.688,406.374,165.556,51.355,159.159
C06158=1020.083,-120.937,406.382,165.553,51.359,159.159
C06159=1020.077,-121.187,406.389,165.550,51.363,159.159
C06160=1020.072,-121.436,406.398,165.547,51.368,159.159
C06161=1020.067,-121.687,406.406,165.544,51.372,159.159
C06162=1020.061,-121.936,406.414,165.541,51.376,159.160
C06163=1020.056,-122.186,406.421,165.538,51.381,159.160
C06164=1020.051,-122.436,406.430,165.535,51.385,159.160
C06165=1020.046,-122.685,406.437,165.532,51.388,159.160
C06166=1020.040,-122.935,406.445,165.528,51.393,159.160
C06167=1020.035,-123.185,406.453,165.526,51.397,159.160
C06168=1020.029,-123.435,406.461,165.523,51.401,159.161
C06169=1020.024,-123.685,406.469,165.519,51.406,159.161
C06170=1020.020,-123.934,406.477,165.517,51.410,159.161
C06171=1020.014,-124.184,406.484,165.514,51.414,159.161
C06172=1020.009,-124.435,406.492,165.510,51.418,159.161
C06173=1020.004,-124.684,406.500,165.507,51.422,159.161
C06174=1019.998,-124.934,406.507,165.505,51.427,159.162
C06175=1019.994,-125.184,406.515,165.501,51.431,159.162
C06176=1019.988,-125.433,406.523,165.499,51.435,159.162
C06177=1019.983,-125.684,406.530,165.495,51.440,159.162
C06178=1019.977,-125.934,406.538,165.492,51.444,159.162
C06179=1019.972,-126.183,406.546,165.490,51.448,159.163
C06180=1019.967,-126.433,406.553,165.486,51.453,159.163
C06181=1019.962,-126.683,406.561,165.483,51.457,159.163
C06182=1019.956,-126.932,406.568,165.481,51.461,159.163
C06183=1019.951,-127.182,406.576,165.477,51.466,159.163
C06184=1019.946,-127.432,406.583,165.475,51.470,159.164
C06185=1019.940,-127.682,406.592,165.472,51.474,159.164
C06186=1019.935,-127.931,406.598,165.468,51.478,159.164
C06187=1019.930,-128.182,406.606,165.465,51.482,159.164
C06188=1019.926,-128.431,406.614,165.462,51.486,159.164
C06189=1019.921,-128.681,406.623,165.459,51.489,159.164
C06190=1019.918,-128.930,406.633,165.457,51.492,159.164
C06191=1019.915,-129.180,406.643,165.454,51.493,159.164
C06192=1019.912,-129.430,406.654,165.451,51.495,159.164
C06193=1019.910,-129.679,406.665,165.449,51.496,159.163
C06194=1019.908,-129.928,406.677,165.446,51.497,159.163
C06195=1019.906,-130.178,406.689,165.444,51.497,159.162
C06196=1019.905,-130.428,406.702,165.442,51.496,159.162
C06197=1019.905,-130.678,406.716,165.439,51.495,159.161
C06198=1019.905,-130.927,406.730,165.437,51.493,159.160
C06199=1019.905,-131.177,406.745,165.435,51.491,159.160
C06200=1019.906,-131.427,406.761,165.433,51.488,159.159
C06201=1019.907,-131.677,406.777,165.431,51.485,159.158
C06202=1019.909,-131.927,406.793,165.429,51.482,159.157
C06203=1019.912,-132.176,406.810,165.427,51.477,159.156
C06204=1019.914,-132.426,406.828,165.426,51.473,159.155
C06205=1019.917,-132.676,406.846,165.424,51.468,159.154
C06206=1019.921,-132.925,406.865,165.422,51.462,159.152
C06207=1019.924,-133.175,406.885,165.420,51.456,159.151
C06208=1019.649,-133.201,406.521,165.377,51.769,159.197
C06209=1019.646,-132.952,406.501,165.378,51.775,159.198
C06210=1019.642,-132.702,406.482,165.380,51.781,159.199
C06211=1019.639,-132.452,406.463,165.381,51.786,159.200
C06212=1019.637,-132.202,406.446,165.384,51.791,159.202
C06213=1019.634,-131.953,406.429,165.385,51.795,159.203
C06214=1019.632,-131.703,406.412,165.387,51.798,159.204
C06215=1019.631,-131.453,406.396,165.389,51.802,159.205
C06216=1019.630,-131.203,406.381,165.392,51.805,159.205
C06217=1019.630,-130.954,406.366,165.394,51.806,159.206
C06218=1019.630,-130.704,406.352,165.396,51.808,159.207
C06219=1019.630,-130.454,406.338,165.398,51.809,159.208
C06220=1019.631,-130.204,406.325,165.400,51.810,159.208
C06221=1019.632,-129.955,406.313,165.403,51.810,159.208
C06222=1019.634,-129.705,406.301,165.405,51.809,159.209
C06223=1019.637,-129.455,406.290,165.407,51.808,159.209
C06224=1019.640,-129.205,406.279,165.410,51.807,159.209
C06225=1019.643,-128.956,406.269,165.413,51.805,159.209
C06226=1019.646,-128.706,406.259,165.416,51.802,159.210
C06227=1019.650,-128.456,406.250,165.418,51.799,159.209
C06228=1019.655,-128.207,406.242,165.421,51.795,159.209
C06229=1019.660,-127.958,406.234,165.425,51.791,159.209
C06230=1019.665,-127.708,406.227,165.428,51.787,159.209
C06231=1019.670,-127.458,406.219,165.430,51.783,159.209
C06232=1019.676,-127.209,406.211,165.434,51.778,159.209
C06233=1019.681,-126.959,406.204,165.436,51.774,159.209
C06234=1019.686,-126.709,406.196,165.439,51.770,159.208
C06235=1019.691,-126.459,406.189,165.443,51.765,159.208
C06236=1019.697,-126.210,406.181,165.445,51.761,159.208
C06237=1019.702,-125.960,406.173,165.449,51.757,159.208
C06238=1019.707,-125.710,406.166,165.451,51.752,159.208
C06239=1019.712,-125.459,406.158,165.455,51.748,159.208
C06240=1019.718,-125.211,406.151,165.458,51.743,159.207
C06241=1019.723,-124.960,406.143,165.460,51.739,159.207
C06242=1019.728,-124.710,406.135,165.464,51.735,159.207
C06243=1019.734,-124.461,406.128,165.466,51.730,159.207
C06244=1019.738,-124.211,406.120,165.470,51.727,159.207
C06245=1019.744,-123.961,406.113,165.473,51.722,159.207
C06246=1019.749,-123.711,406.104,165.476,51.718,159.206
C06247=1019.754,-123.461,406.097,165.479,51.714,159.206
C06248=1019.760,-123.211,406.089,165.482,51.709,159.206
C06249=1019.764,-122.962,406.081,165.484,51.705,159.206
C06250=1019.769,-122.711,406.074,165.488,51.700,159.206
C06251=1019.775,-122.462,406.066,165.491,51.696,159.205
C06252=1019.780,-122.212,406.058,165.494,51.692,159.205
C06253=1019.785,-121.962,406.049,165.497,51.687,159.205
C06254=1019.791,-121.713,406.043,165.499,51.683,159.205
C06255=1019.796,-121.463,406.034,165.503,51.679,159.205
C06256=1019.801,-121.213,406.026,165.506,51.675,159.205
C06257=1019.807,-120.963,406.019,165.510,51.671,159.204
C06258=1019.812,-120.713,406.011,165.512,51.666,159.204
C06259=1019.817,-120.463,406.002,165.515,51.662,159.204
C06260=1019.821,-120.214,405.995,165.518,51.658,159.204
C06261=1019.827,-119.964,405.987,165.521,51.653,159.204
C06262=1019.832,-119.714,405.979,165.524,51.649,159.203
C06263=1019.838,-119.464,405.971,165.527,51.645,159.203
C06264=1019.843,-119.214,405.964,165.530,51.640,159.203
C06265=1019.849,-118.964,405.955,165.533,51.636,159.203
C06266=1019.854,-118.715,405.947,165.536,51.632,159.203
C06267=1019.860,-118.465,405.939,165.540,51.627,159.203
C06268=1019.864,-118.216,405.931,165.542,51.623,159.202
C06269=1019.870,-117.931,405.922,165.546,51.618,159.202
C06270=1019.876,-117.647,405.913,165.549,51.613,159.202
C06271=1019.882,-117.363,405.904,165.553,51.608,159.202
C06272=1019.889,-117.078,405.894,165.556,51.603,159.201
///RCONF 1,0,0,0,0,0,0,0,0,0,0,0,0,0,0,0,0,0,0,0,0,0,0,0
C06273=1019.894,-116.828,405.887,165.559,51.599,159.201
C06274=1019.899,-116.578,405.878,165.562,51.594,159.201
C06275=1019.904,-116.329,405.870,165.565,51.591,159.201
C06276=1019.909,-116.079,405.863,165.569,51.586,159.201
C06277=1019.915,-115.829,405.854,165.571,51.582,159.201
C06278=1019.920,-115.579,405.846,165.574,51.578,159.200
C06279=1019.925,-115.330,405.837,165.578,51.573,159.200
C06280=1019.931,-115.080,405.830,165.580,51.569,159.200
C06281=1019.936,-114.830,405.822,165.584,51.564,159.200
C06282=1019.941,-114.580,405.813,165.586,51.560,159.200
C06283=1019.946,-114.330,405.806,165.590,51.556,159.199
C06284=1019.952,-114.080,405.797,165.593,51.551,159.199
C06285=1019.957,-113.830,405.789,165.595,51.547,159.199
C06286=1019.962,-113.581,405.780,165.599,51.543,159.199
C06287=1019.968,-113.331,405.772,165.602,51.538,159.199
C06288=1019.973,-113.081,405.764,165.605,51.534,159.198
C06289=1019.978,-112.831,405.756,165.608,51.530,159.198
C06290=1019.984,-112.582,405.747,165.610,51.525,159.198
C06291=1019.989,-112.332,405.739,165.614,51.521,159.198
C06292=1019.994,-112.082,405.730,165.617,51.517,159.198
C06293=1019.999,-111.832,405.722,165.621,51.513,159.198
C06294=1020.005,-111.583,405.714,165.623,51.509,159.197
C06295=1020.010,-111.332,405.706,165.626,51.504,159.197
C06296=1020.016,-111.082,405.697,165.629,51.500,159.197
C06297=1020.021,-110.833,405.689,165.632,51.496,159.197
C06298=1020.027,-110.583,405.681,165.636,51.491,159.197
C06299=1020.032,-110.333,405.672,165.638,51.487,159.196
C06300=1020.037,-110.083,405.664,165.642,51.482,159.196
C06301=1020.043,-109.834,405.655,165.645,51.478,159.196
C06302=1020.048,-109.584,405.647,165.647,51.474,159.196
C06303=1020.053,-109.334,405.638,165.651,51.469,159.196
C06304=1020.058,-109.085,405.630,165.653,51.465,159.195
C06305=1020.064,-108.835,405.621,165.657,51.461,159.195
C06306=1020.069,-108.585,405.613,165.660,51.456,159.195
C06307=1020.075,-108.335,405.604,165.663,51.452,159.195
C06308=1020.081,-108.085,405.596,165.666,51.448,159.195
C06309=1020.086,-107.836,405.587,165.668,51.444,159.194
C06310=1020.091,-107.586,405.579,165.672,51.439,159.194
C06311=1020.097,-107.336,405.570,165.675,51.435,159.194
C06312=1020.102,-107.086,405.562,165.678,51.430,159.194
C06313=1020.106,-106.836,405.553,165.681,51.426,159.194
C06314=1020.112,-106.586,405.544,165.684,51.422,159.193
C06315=1020.117,-106.336,405.536,165.687,51.417,159.193
C06316=1020.123,-106.087,405.527,165.690,51.413,159.193
C06317=1020.128,-105.837,405.519,165.694,51.409,159.193
C06318=1020.133,-105.587,405.510,165.696,51.405,159.193
C06319=1020.138,-105.337,405.502,165.699,51.401,159.193
C06320=1020.144,-105.087,405.493,165.703,51.396,159.192
C06321=1020.150,-104.838,405.484,165.705,51.392,159.192
C06322=1020.155,-104.588,405.475,165.709,51.388,159.192
C06323=1020.160,-104.338,405.467,165.711,51.383,159.192
C06324=1020.166,-104.089,405.458,165.714,51.379,159.191
C06325=1020.172,-103.838,405.449,165.718,51.375,159.191
C06326=1020.176,-103.589,405.439,165.720,51.370,159.191
C06327=1020.182,-103.339,405.431,165.724,51.366,159.191
C06328=1020.187,-103.089,405.422,165.727,51.362,159.191
C06329=1020.193,-102.839,405.414,165.730,51.357,159.191
C06330=1020.198,-102.589,405.405,165.733,51.353,159.190
C06331=1020.204,-102.340,405.396,165.735,51.349,159.190
C06332=1020.209,-102.091,405.387,165.739,51.344,159.190
C06333=1020.215,-101.806,405.377,165.743,51.340,159.190
C06334=1020.221,-101.521,405.367,165.746,51.335,159.189
C06335=1020.228,-101.237,405.357,165.750,51.330,159.189
C06336=1020.234,-100.953,405.347,165.753,51.325,159.189
C06337=1020.239,-100.703,405.338,165.756,51.321,159.189
C06338=1020.244,-100.453,405.329,165.759,51.316,159.189
C06339=1020.249,-100.203,405.320,165.762,51.312,159.188
C06340=1020.255,-99.953,405.311,165.765,51.307,159.188
C06341=1020.261,-99.704,405.302,165.768,51.303,159.188
C06342=1020.266,-99.454,405.294,165.772,51.299,159.188
C06343=1020.272,-99.204,405.284,165.774,51.294,159.188
C06344=1020.277,-98.954,405.276,165.777,51.290,159.187
C06345=1020.282,-98.704,405.267,165.781,51.286,159.187
C06346=1020.288,-98.455,405.257,165.783,51.282,159.187
C06347=1020.293,-98.205,405.249,165.787,51.277,159.187
C06348=1020.299,-97.956,405.240,165.789,51.273,159.187
C06349=1020.305,-97.705,405.231,165.793,51.268,159.186
C06350=1020.310,-97.456,405.221,165.796,51.264,159.186
C06351=1020.315,-97.206,405.212,165.799,51.261,159.186
C06352=1020.320,-96.955,405.203,165.802,51.256,159.186
C06353=1020.325,-96.706,405.194,165.805,51.252,159.186
C06354=1020.332,-96.457,405.184,165.808,51.248,159.185
C06355=1020.336,-96.207,405.175,165.811,51.243,159.185
C06356=1020.342,-95.957,405.166,165.814,51.239,159.185
C06357=1020.347,-95.707,405.156,165.817,51.236,159.185
C06358=1020.352,-95.458,405.147,165.820,51.231,159.185
C06359=1020.358,-95.207,405.138,165.823,51.227,159.185
C06360=1020.363,-94.958,405.129,165.827,51.222,159.184
C06361=1020.369,-94.709,405.119,165.829,51.218,159.184
C06362=1020.374,-94.458,405.110,165.832,51.214,159.184
C06363=1020.379,-94.209,405.101,165.836,51.209,159.184
C06364=1020.385,-93.958,405.091,165.838,51.205,159.183
C06365=1020.390,-93.709,405.082,165.841,51.201,159.183
C06366=1020.396,-93.459,405.073,165.845,51.197,159.183
C06367=1020.401,-93.209,405.064,165.847,51.193,159.183
C06368=1020.406,-92.960,405.054,165.851,51.189,159.183
C06369=1020.412,-92.710,405.044,165.854,51.184,159.183
C06370=1020.417,-92.460,405.036,165.856,51.180,159.182
C06371=1020.423,-92.210,405.025,165.860,51.176,159.182
C06372=1020.428,-91.961,405.016,165.863,51.172,159.182
C06373=1020.434,-91.711,405.007,165.865,51.167,159.182
C06374=1020.439,-91.461,404.998,165.869,51.163,159.182
C06375=1020.445,-91.212,404.988,165.872,51.159,159.181
C06376=1020.449,-90.961,404.979,165.875,51.154,159.181
C06377=1020.456,-90.712,404.969,165.878,51.150,159.181
C06378=1020.460,-90.462,404.960,165.880,51.146,159.181
C06379=1020.467,-90.212,404.950,165.884,51.141,159.180
C06380=1020.472,-89.963,404.942,165.887,51.137,159.180
C06381=1020.477,-89.713,404.931,165.891,51.133,159.180
C06382=1020.483,-89.464,404.922,165.893,51.129,159.180
C06383=1020.488,-89.213,404.912,165.896,51.125,159.180
C06384=1020.494,-88.964,404.903,165.900,51.121,159.180
C06385=1020.499,-88.714,404.893,165.902,51.116,159.179
C06386=1020.505,-88.464,404.884,165.906,51.112,159.179
C06387=1020.510,-88.214,404.874,165.909,51.108,159.179
C06388=1020.516,-87.965,404.864,165.912,51.103,159.179
C06389=1020.521,-87.715,404.855,165.915,51.099,159.178
C06390=1020.527,-87.465,404.846,165.917,51.095,159.178
C06391=1020.533,-87.216,404.837,165.921,51.090,159.178
C06392=1020.538,-86.966,404.826,165.924,51.086,159.178
C06393=1020.544,-86.716,404.817,165.927,51.082,159.178
C06394=1020.549,-86.466,404.807,165.930,51.077,159.177
C06395=1020.555,-86.217,404.798,165.933,51.072,159.177
C06396=1020.560,-85.967,404.788,165.936,51.068,159.177
C06397=1020.566,-85.684,404.777,165.940,51.064,159.177
C06398=1020.573,-85.402,404.766,165.943,51.058,159.176
C06399=1020.578,-85.120,404.756,165.946,51.054,159.176
C06400=1020.585,-84.838,404.744,165.950,51.049,159.176
C06401=1020.591,-84.588,404.735,165.952,51.045,159.176
C06402=1020.597,-84.339,404.725,165.956,51.040,159.175
C06403=1020.602,-84.089,404.715,165.959,51.036,159.175
C06404=1020.608,-83.839,404.706,165.962,51.031,159.175
C06405=1020.613,-83.589,404.696,165.965,51.027,159.175
C06406=1020.619,-83.340,404.686,165.969,51.023,159.175
C06407=1020.625,-83.089,404.676,165.971,51.019,159.174
C06408=1020.630,-82.840,404.667,165.975,51.013,159.174
C06409=1020.636,-82.590,404.657,165.977,51.009,159.174
C06410=1020.642,-82.340,404.647,165.980,51.005,159.173
C06411=1020.647,-82.090,404.637,165.983,51.001,159.173
C06412=1020.653,-81.841,404.628,165.986,50.996,159.173
C06413=1020.658,-81.591,404.618,165.990,50.992,159.173
C06414=1020.665,-81.341,404.608,165.992,50.988,159.173
C06415=1020.669,-81.092,404.598,165.996,50.983,159.172
C06416=1020.676,-80.842,404.589,165.999,50.979,159.172
C06417=1020.681,-80.592,404.579,166.002,50.974,159.172
C06418=1020.687,-80.342,404.569,166.005,50.970,159.171
C06419=1020.692,-80.093,404.559,166.008,50.965,159.171
C06420=1020.697,-79.843,404.549,166.011,50.961,159.171
C06421=1020.704,-79.593,404.540,166.013,50.957,159.171
C06422=1020.709,-79.343,404.529,166.017,50.952,159.171
C06423=1020.714,-79.094,404.519,166.020,50.948,159.170
C06424=1020.720,-78.844,404.509,166.022,50.944,159.170
C06425=1020.726,-78.594,404.499,166.026,50.940,159.170
C06426=1020.731,-78.344,404.489,166.029,50.936,159.170
C06427=1020.737,-78.094,404.479,166.033,50.932,159.170
C06428=1020.743,-77.845,404.469,166.035,50.928,159.169
C06429=1020.748,-77.595,404.459,166.038,50.923,159.169
C06430=1020.753,-77.345,404.449,166.042,50.919,159.169
C06431=1020.759,-77.096,404.438,166.044,50.915,159.169
C06432=1020.764,-76.846,404.428,166.047,50.911,159.168
C06433=1020.770,-76.596,404.418,166.051,50.906,159.168
C06434=1020.776,-76.346,404.408,166.053,50.902,159.168
C06435=1020.781,-76.097,404.397,166.057,50.898,159.168
C06436=1020.787,-75.847,404.387,166.060,50.893,159.168
C06437=1020.793,-75.597,404.378,166.062,50.889,159.167
C06438=1020.798,-75.348,404.367,166.066,50.885,159.167
C06439=1020.804,-75.098,404.357,166.068,50.880,159.167
C06440=1020.809,-74.848,404.347,166.072,50.875,159.167
C06441=1020.815,-74.599,404.337,166.074,50.871,159.166
C06442=1020.821,-74.349,404.326,166.077,50.867,159.166
C06443=1020.826,-74.099,404.316,166.081,50.863,159.166
C06444=1020.832,-73.849,404.305,166.084,50.859,159.166
C06445=1020.837,-73.599,404.295,166.086,50.855,159.165
C06446=1020.843,-73.350,404.285,166.090,50.851,159.165
C06447=1020.847,-73.100,404.274,166.093,50.847,159.165
C06448=1020.853,-72.850,404.263,166.095,50.842,159.165
C06449=1020.858,-72.600,404.253,166.098,50.839,159.165
C06450=1020.864,-72.351,404.242,166.102,50.834,159.165
C06451=1020.870,-72.101,404.231,166.105,50.830,159.164
C06452=1020.875,-71.851,404.221,166.107,50.826,159.164
C06453=1020.881,-71.602,404.210,166.111,50.822,159.164
C06454=1020.886,-71.352,404.200,166.114,50.818,159.164
C06455=1020.892,-71.103,404.189,166.116,50.813,159.163
C06456=1020.897,-70.853,404.179,166.120,50.809,159.163
C06457=1020.903,-70.603,404.168,166.123,50.806,159.163
C06458=1020.909,-70.354,404.157,166.125,50.801,159.163
C06459=1020.914,-70.103,404.147,166.129,50.797,159.163
C06460=1020.920,-69.854,404.136,166.132,50.793,159.162
C06461=1020.926,-69.573,404.125,166.135,50.788,159.162
C06462=1020.932,-69.293,404.113,166.139,50.783,159.162
C06463=1020.939,-69.013,404.100,166.141,50.779,159.162
C06464=1020.944,-68.733,404.089,166.145,50.774,159.161
C06465=1020.950,-68.483,404.078,166.148,50.769,159.161
C06466=1020.956,-68.233,404.068,166.151,50.765,159.161
C06467=1020.961,-67.984,404.057,166.154,50.761,159.160
C06468=1020.966,-67.734,404.046,166.157,50.757,159.160
C06469=1020.972,-67.485,404.035,166.160,50.753,159.160
C06470=1020.977,-67.234,404.025,166.163,50.749,159.160
C06471=1020.983,-66.985,404.014,166.167,50.745,159.160
C06472=1020.989,-66.735,404.003,166.169,50.741,159.159
C06473=1020.994,-66.485,403.993,166.172,50.736,159.159
C06474=1021.000,-66.236,403.982,166.176,50.732,159.159
C06475=1021.006,-65.986,403.971,166.178,50.728,159.159
C06476=1021.012,-65.737,403.960,166.181,50.724,159.158
C06477=1021.017,-65.487,403.950,166.185,50.719,159.158
C06478=1021.022,-65.237,403.938,166.187,50.715,159.158
C06479=1021.028,-64.987,403.928,166.190,50.711,159.158
C06480=1021.034,-64.737,403.916,166.194,50.707,159.158
C06481=1021.039,-64.487,403.906,166.196,50.702,159.157
C06482=1021.045,-64.238,403.895,166.199,50.698,159.157
C06483=1021.051,-63.988,403.884,166.203,50.694,159.157
C06484=1021.057,-63.739,403.874,166.205,50.690,159.157
C06485=1021.062,-63.489,403.863,166.208,50.686,159.156
C06486=1021.068,-63.239,403.852,166.211,50.681,159.156
C06487=1021.074,-62.990,403.842,166.214,50.677,159.156
C06488=1021.079,-62.740,403.831,166.217,50.673,159.156
C06489=1021.084,-62.490,403.819,166.220,50.668,159.155
C06490=1021.090,-62.241,403.808,166.223,50.664,159.155
C06491=1021.096,-61.991,403.797,166.225,50.659,159.155
C06492=1021.102,-61.741,403.786,166.229,50.655,159.154
C06493=1021.108,-61.491,403.776,166.232,50.651,159.154
C06494=1021.113,-61.242,403.765,166.235,50.646,159.154
C06495=1021.119,-60.992,403.754,166.238,50.642,159.154
C06496=1021.125,-60.743,403.743,166.241,50.638,159.153
C06497=1021.131,-60.493,403.733,166.244,50.634,159.153
C06498=1021.136,-60.243,403.721,166.247,50.630,159.153
C06499=1021.142,-59.993,403.710,166.250,50.625,159.153
C06500=1021.148,-59.744,403.699,166.253,50.621,159.153
C06501=1021.153,-59.494,403.688,166.256,50.617,159.152
C06502=1021.159,-59.245,403.677,166.258,50.612,159.152
C06503=1021.165,-58.995,403.666,166.262,50.608,159.152
C06504=1021.171,-58.745,403.655,166.265,50.604,159.151
C06505=1021.177,-58.495,403.644,166.268,50.599,159.151
C06506=1021.182,-58.245,403.633,166.271,50.595,159.151
C06507=1021.187,-57.996,403.623,166.274,50.591,159.151
C06508=1021.193,-57.746,403.612,166.277,50.586,159.150
C06509=1021.199,-57.496,403.600,166.280,50.582,159.150
C06510=1021.205,-57.246,403.590,166.283,50.577,159.150
C06511=1021.211,-56.998,403.578,166.286,50.573,159.150
C06512=1021.217,-56.748,403.567,166.288,50.569,159.149
C06513=1021.223,-56.498,403.556,166.292,50.564,159.149
C06514=1021.228,-56.248,403.544,166.295,50.560,159.149
C06515=1021.234,-55.999,403.534,166.297,50.556,159.148
C06516=1021.240,-55.749,403.523,166.301,50.551,159.148
C06517=1021.246,-55.499,403.511,166.303,50.547,159.148
C06518=1021.252,-55.249,403.501,166.307,50.543,159.148
C06519=1021.258,-55.000,403.490,166.310,50.538,159.147
C06520=1021.264,-54.750,403.478,166.312,50.534,159.147
C06521=1021.269,-54.500,403.467,166.316,50.529,159.147
C06522=1021.275,-54.250,403.456,166.318,50.525,159.146
C06523=1021.280,-54.001,403.445,166.322,50.521,159.146
C06524=1021.287,-53.751,403.434,166.325,50.517,159.146
C06525=1021.293,-53.472,403.421,166.328,50.511,159.146
C06526=1021.300,-53.193,403.409,166.331,50.506,159.145
C06527=1021.306,-52.914,403.396,166.335,50.502,159.145
C06528=1021.313,-52.635,403.384,166.338,50.497,159.145
C06529=1021.319,-52.385,403.372,166.341,50.493,159.144
C06530=1021.325,-52.135,403.362,166.343,50.488,159.144
C06531=1021.331,-51.886,403.351,166.347,50.483,159.144
C06532=1021.337,-51.636,403.339,166.350,50.479,159.143
C06533=1021.342,-51.387,403.327,166.353,50.475,159.143
C06534=1021.348,-51.137,403.316,166.356,50.470,159.143
C06535=1021.354,-50.887,403.305,166.359,50.466,159.143
C06536=1021.359,-50.637,403.294,166.362,50.461,159.142
C06537=1021.366,-50.388,403.282,166.365,50.457,159.142
C06538=1021.371,-50.138,403.270,166.367,50.453,159.142
C06539=1021.377,-49.888,403.259,166.371,50.449,159.142
C06540=1021.383,-49.638,403.247,166.374,50.445,159.141
C06541=1021.388,-49.389,403.236,166.376,50.441,159.141
C06542=1021.394,-49.140,403.224,166.379,50.437,159.141
C06543=1021.400,-48.890,403.212,166.383,50.432,159.141
C06544=1021.405,-48.640,403.200,166.385,50.428,159.140
C06545=1021.412,-48.390,403.189,166.388,50.424,159.140
C06546=1021.417,-48.140,403.178,166.392,50.420,159.140
C06547=1021.423,-47.891,403.166,166.394,50.415,159.140
C06548=1021.428,-47.641,403.154,166.397,50.411,159.139
C06549=1021.434,-47.392,403.142,166.400,50.407,159.139
C06550=1021.440,-47.142,403.131,166.403,50.403,159.139
C06551=1021.445,-46.892,403.118,166.406,50.399,159.138
C06552=1021.451,-46.643,403.108,166.409,50.395,159.138
C06553=1021.457,-46.393,403.095,166.411,50.391,159.138
C06554=1021.463,-46.144,403.084,166.415,50.386,159.138
C06555=1021.469,-45.894,403.072,166.418,50.382,159.137
C06556=1021.474,-45.644,403.061,166.420,50.378,159.137
C06557=1021.479,-45.429,403.050,166.423,50.374,159.137
C06558=1021.484,-45.214,403.040,166.426,50.370,159.137
C06559=1021.489,-44.999,403.030,166.428,50.367,159.136
C06560=1021.494,-44.785,403.020,166.430,50.363,159.136
C06561=1021.499,-44.570,403.010,166.433,50.359,159.136
C06562=1021.504,-44.356,403.000,166.435,50.355,159.135
C06563=1021.508,-44.140,402.989,166.438,50.352,159.135
C06564=1021.514,-43.925,402.979,166.441,50.348,159.135
C06565=1021.520,-43.676,402.968,166.443,50.344,159.135
C06566=1021.526,-43.427,402.955,166.446,50.340,159.135
C06567=1021.531,-43.177,402.944,166.450,50.335,159.134
C06568=1021.537,-42.927,402.932,166.452,50.331,159.134
C06569=1021.542,-42.677,402.920,166.455,50.327,159.134
C06570=1021.549,-42.428,402.908,166.459,50.323,159.134
C06571=1021.554,-42.179,402.896,166.461,50.318,159.133
C06572=1021.561,-41.928,402.885,166.464,50.314,159.133
C06573=1021.566,-41.679,402.873,166.467,50.309,159.133
C06574=1021.573,-41.430,402.861,166.470,50.305,159.132
C06575=1021.578,-41.180,402.849,166.473,50.301,159.132
C06576=1021.584,-40.930,402.837,166.476,50.297,159.132
C06577=1021.590,-40.681,402.825,166.479,50.292,159.131
C06578=1021.595,-40.431,402.813,166.481,50.288,159.131
C06579=1021.602,-40.181,402.801,166.484,50.284,159.131
C06580=1021.607,-39.932,402.789,166.488,50.279,159.131
C06581=1021.614,-39.682,402.778,166.490,50.275,159.130
C06582=1021.619,-39.433,402.766,166.493,50.271,159.130
C06583=1021.625,-39.183,402.753,166.496,50.266,159.130
C06584=1021.630,-38.933,402.741,166.499,50.262,159.129
C06585=1021.636,-38.683,402.730,166.502,50.258,159.129
C06586=1021.642,-38.433,402.717,166.504,50.254,159.129
C06587=1021.648,-38.184,402.705,166.508,50.250,159.129
C06588=1021.653,-37.934,402.692,166.511,50.245,159.128
C06589=1021.662,-37.586,402.675,166.515,50.239,159.128
C06590=1021.670,-37.238,402.659,166.519,50.234,159.128
C06591=1021.677,-36.889,402.641,166.523,50.228,159.127
C06592=1021.685,-36.541,402.624,166.526,50.222,159.127
C06593=1021.691,-36.291,402.612,166.530,50.218,159.126
C06594=1021.697,-36.041,402.599,166.533,50.214,159.126
C06595=1021.702,-35.792,402.587,166.535,50.209,159.126
C06596=1021.709,-35.542,402.575,166.538,50.205,159.125
C06597=1021.715,-35.292,402.563,166.542,50.201,159.125
C06598=1021.720,-35.042,402.551,166.544,50.197,159.125
C06599=1021.726,-34.793,402.538,166.547,50.193,159.125
C06600=1021.732,-34.543,402.526,166.550,50.189,159.124
C06601=1021.737,-34.293,402.514,166.553,50.184,159.124
C06602=1021.743,-34.044,402.501,166.556,50.180,159.124
C06603=1021.750,-33.794,402.489,166.558,50.176,159.123
C06604=1021.755,-33.545,402.477,166.561,50.171,159.123
C06605=1021.761,-33.295,402.464,166.565,50.167,159.123
C06606=1021.767,-33.045,402.452,166.567,50.163,159.123
C06607=1021.772,-32.796,402.440,166.570,50.159,159.122
C06608=1021.778,-32.546,402.427,166.573,50.155,159.122
C06609=1021.784,-32.296,402.414,166.576,50.150,159.122
C06610=1021.791,-32.047,402.403,166.579,50.146,159.121
C06611=1021.796,-31.797,402.390,166.581,50.142,159.121
C06612=1021.802,-31.547,402.378,166.584,50.138,159.121
C06613=1021.808,-31.298,402.365,166.588,50.133,159.121
C06614=1021.814,-31.048,402.352,166.590,50.129,159.120
C06615=1021.819,-30.799,402.340,166.593,50.125,159.120
C06616=1021.825,-30.549,402.327,166.595,50.120,159.119
C06617=1021.832,-30.300,402.315,166.599,50.116,159.119
C06618=1021.838,-30.050,402.303,166.602,50.112,159.119
C06619=1021.843,-29.801,402.291,166.604,50.108,159.119
C06620=1021.849,-29.551,402.278,166.607,50.104,159.118
C06621=1021.855,-29.301,402.265,166.611,50.099,159.118
C06622=1021.861,-29.051,402.253,166.613,50.095,159.118
C06623=1021.866,-28.802,402.241,166.616,50.090,159.117
C06624=1021.872,-28.553,402.227,166.619,50.086,159.117
C06625=1021.878,-28.303,402.215,166.622,50.081,159.117
C06626=1021.885,-28.053,402.203,166.625,50.077,159.116
C06627=1021.891,-27.803,402.190,166.627,50.073,159.116
C06628=1021.896,-27.554,402.178,166.630,50.069,159.116
C06629=1021.902,-27.304,402.166,166.634,50.065,159.116
C06630=1021.908,-27.055,402.152,166.636,50.061,159.115
C06631=1021.913,-26.805,402.139,166.639,50.056,159.115
C06632=1021.919,-26.555,402.127,166.641,50.052,159.114
C06633=1021.925,-26.305,402.114,166.644,50.048,159.114
C06634=1021.931,-26.056,402.101,166.648,50.043,159.114
C06635=1021.937,-25.806,402.089,166.650,50.039,159.114
C06636=1021.943,-25.557,402.076,166.653,50.035,159.113
C06637=1021.948,-25.307,402.062,166.656,50.031,159.113
C06638=1021.954,-25.057,402.050,166.658,50.027,159.113
C06639=1021.960,-24.807,402.037,166.661,50.023,159.112
C06640=1021.966,-24.558,402.024,166.665,50.019,159.112
C06641=1021.971,-24.309,402.012,166.668,50.015,159.112
C06642=1021.978,-24.060,401.998,166.670,50.010,159.111
C06643=1021.983,-23.810,401.986,166.673,50.006,159.111
C06644=1021.989,-23.559,401.973,166.675,50.002,159.111
C06645=1021.995,-23.310,401.959,166.679,49.997,159.111
C06646=1022.001,-23.060,401.947,166.682,49.993,159.110
C06647=1022.007,-22.811,401.934,166.684,49.989,159.110
C06648=1022.012,-22.562,401.921,166.687,49.985,159.110
C06649=1022.018,-22.312,401.909,166.689,49.981,159.109
C06650=1022.024,-22.062,401.895,166.692,49.976,159.109
C06651=1022.030,-21.813,401.882,166.696,49.972,159.109
C06652=1022.036,-21.563,401.869,166.698,49.968,159.108
C06653=1022.042,-21.284,401.855,166.702,49.963,159.108
C06654=1022.049,-21.004,401.840,166.704,49.959,159.108
C06655=1022.056,-20.724,401.826,166.708,49.954,159.107
C06656=1022.062,-20.445,401.811,166.711,49.949,159.107
C06657=1022.068,-20.195,401.799,166.714,49.945,159.107
C06658=1022.074,-19.946,401.785,166.717,49.941,159.106
C06659=1022.080,-19.696,401.772,166.719,49.937,159.106
C06660=1022.086,-19.446,401.759,166.722,49.932,159.106
C06661=1022.092,-19.197,401.746,166.725,49.928,159.105
C06662=1022.098,-18.947,401.733,166.728,49.924,159.105
C06663=1022.104,-18.697,401.721,166.731,49.919,159.105
C06664=1022.109,-18.448,401.707,166.733,49.915,159.104
C06665=1022.115,-18.198,401.694,166.736,49.911,159.104
C06666=1022.121,-17.949,401.681,166.739,49.906,159.104
C06667=1022.127,-17.699,401.668,166.742,49.902,159.103
C06668=1022.134,-17.450,401.655,166.744,49.898,159.103
C06669=1022.139,-17.199,401.642,166.747,49.893,159.103
C06670=1022.145,-16.950,401.629,166.751,49.889,159.102
C06671=1022.151,-16.701,401.615,166.754,49.885,159.102
C06672=1022.157,-16.451,401.603,166.756,49.880,159.102
C06673=1022.163,-16.202,401.589,166.759,49.876,159.101
C06674=1022.169,-15.952,401.577,166.761,49.872,159.101
C06675=1022.175,-15.702,401.563,166.765,49.868,159.101
C06676=1022.181,-15.453,401.550,166.767,49.863,159.100
C06677=1022.186,-15.203,401.536,166.770,49.859,159.100
C06678=1022.192,-14.954,401.523,166.773,49.855,159.100
C06679=1022.198,-14.704,401.510,166.775,49.851,159.099
C06680=1022.204,-14.455,401.496,166.778,49.847,159.099
C06681=1022.210,-14.205,401.483,166.781,49.843,159.099
C06682=1022.215,-13.955,401.470,166.783,49.839,159.098
C06683=1022.222,-13.706,401.457,166.787,49.835,159.098
C06684=1022.227,-13.456,401.443,166.790,49.830,159.098
C06685=1022.233,-13.207,401.429,166.792,49.826,159.097
C06686=1022.238,-12.957,401.416,166.795,49.822,159.097
C06687=1022.245,-12.708,401.403,166.798,49.818,159.097
C06688=1022.250,-12.458,401.389,166.800,49.814,159.097
C06689=1022.257,-12.208,401.375,166.803,49.810,159.096
C06690=1022.262,-11.959,401.362,166.806,49.805,159.096
C06691=1022.269,-11.709,401.348,166.809,49.801,159.096
C06692=1022.274,-11.459,401.335,166.812,49.797,159.095
C06693=1022.280,-11.210,401.322,166.814,49.793,159.095
C06694=1022.286,-10.961,401.309,166.817,49.788,159.095
C06695=1022.292,-10.711,401.295,166.820,49.784,159.094
C06696=1022.298,-10.462,401.282,166.822,49.780,159.094
C06697=1022.303,-10.212,401.268,166.825,49.776,159.093
C06698=1022.310,-9.963,401.254,166.829,49.771,159.093
C06699=1022.315,-9.712,401.241,166.831,49.767,159.093
C06700=1022.322,-9.463,401.228,166.834,49.763,159.092
C06701=1022.327,-9.213,401.214,166.836,49.759,159.092
C06702=1022.333,-8.964,401.200,166.839,49.755,159.092
C06703=1022.339,-8.714,401.187,166.842,49.750,159.092
C06704=1022.345,-8.465,401.173,166.845,49.745,159.091
C06705=1022.350,-8.215,401.159,166.848,49.741,159.091
C06706=1022.357,-7.965,401.146,166.851,49.737,159.091
C06707=1022.363,-7.716,401.132,166.853,49.733,159.090
C06708=1022.369,-7.467,401.119,166.856,49.729,159.090
C06709=1022.374,-7.217,401.105,166.858,49.725,159.089
C06710=1022.381,-6.968,401.092,166.861,49.721,159.089
C06711=1022.387,-6.719,401.078,166.865,49.716,159.089
C06712=1022.393,-6.468,401.064,166.867,49.712,159.088
C06713=1022.399,-6.219,401.051,166.870,49.707,159.088
C06714=1022.405,-5.969,401.037,166.873,49.703,159.088
C06715=1022.411,-5.720,401.024,166.875,49.699,159.087
C06716=1022.416,-5.471,401.010,166.878,49.695,159.087
C06717=1022.423,-5.189,400.995,166.881,49.690,159.087
C06718=1022.430,-4.908,400.979,166.884,49.685,159.086
C06719=1022.436,-4.626,400.964,166.887,49.680,159.086
C06720=1022.443,-4.345,400.948,166.890,49.676,159.085
C06721=1022.450,-4.095,400.935,166.893,49.671,159.085
C06722=1022.456,-3.845,400.921,166.895,49.667,159.085
C06723=1022.461,-3.596,400.907,166.898,49.663,159.084
C06724=1022.467,-3.346,400.893,166.901,49.659,159.084
C06725=1022.473,-3.097,400.878,166.905,49.655,159.084
C06726=1022.478,-2.847,400.864,166.907,49.650,159.083
C06727=1022.484,-2.597,400.850,166.910,49.646,159.083
C06728=1022.490,-2.348,400.837,166.913,49.642,159.083
C06729=1022.496,-2.099,400.823,166.915,49.638,159.082
C06730=1022.502,-1.849,400.808,166.918,49.634,159.082
C06731=1022.507,-1.599,400.794,166.921,49.630,159.082
C06732=1022.513,-1.350,400.781,166.923,49.626,159.081
C06733=1022.519,-1.101,400.766,166.926,49.622,159.081
C06734=1022.526,-0.851,400.752,166.929,49.618,159.081
C06735=1022.531,-0.601,400.739,166.931,49.614,159.080
C06736=1022.537,-0.352,400.725,166.934,49.609,159.080
C06737=1022.543,-0.102,400.710,166.936,49.605,159.080
C06738=1022.548,0.148,400.696,166.939,49.601,159.079
C06739=1022.554,0.397,400.682,166.942,49.597,159.079
C06740=1022.560,0.646,400.667,166.945,49.593,159.079
C06741=1022.566,0.896,400.654,166.947,49.589,159.078
C06742=1022.572,1.146,400.640,166.950,49.584,159.078
C06743=1022.578,1.395,400.625,166.953,49.580,159.078
C06744=1022.584,1.645,400.611,166.956,49.576,159.077
C06745=1022.589,1.894,400.597,166.959,49.572,159.077
C06746=1022.595,2.143,400.583,166.961,49.568,159.077
C06747=1022.601,2.394,400.568,166.964,49.563,159.076
C06748=1022.607,2.643,400.555,166.967,49.559,159.076
C06749=1022.613,2.892,400.541,166.969,49.555,159.076
C06750=1022.619,3.142,400.526,166.972,49.551,159.075
C06751=1022.625,3.391,400.512,166.974,49.546,159.075
C06752=1022.630,3.641,400.498,166.977,49.542,159.074
C06753=1022.637,3.891,400.484,166.980,49.538,159.074
C06754=1022.642,4.140,400.469,166.982,49.534,159.074
C06755=1022.649,4.389,400.456,166.985,49.530,159.073
C06756=1022.655,4.639,400.441,166.988,49.526,159.073
C06757=1022.660,4.888,400.427,166.991,49.521,159.073
C06758=1022.666,5.137,400.412,166.994,49.517,159.072
C06759=1022.672,5.388,400.398,166.996,49.513,159.072
C06760=1022.678,5.637,400.384,166.999,49.509,159.072
C06761=1022.684,5.887,400.369,167.002,49.505,159.071
C06762=1022.690,6.136,400.356,167.004,49.500,159.071
C06763=1022.696,6.385,400.342,167.007,49.496,159.070
C06764=1022.702,6.635,400.327,167.010,49.492,159.070
C06765=1022.708,6.884,400.313,167.012,49.488,159.070
C06766=1022.714,7.135,400.298,167.015,49.483,159.069
C06767=1022.720,7.384,400.284,167.017,49.479,159.069
C06768=1022.725,7.633,400.270,167.020,49.475,159.069
C06769=1022.732,7.883,400.255,167.024,49.470,159.068
C06770=1022.738,8.132,400.242,167.026,49.466,159.068
C06771=1022.744,8.382,400.227,167.029,49.462,159.068
C06772=1022.750,8.631,400.213,167.031,49.458,159.067
C06773=1022.756,8.881,400.198,167.034,49.454,159.067
C06774=1022.762,9.130,400.183,167.036,49.449,159.066
C06775=1022.768,9.380,400.169,167.039,49.445,159.066
C06776=1022.774,9.629,400.155,167.042,49.441,159.066
C06777=1022.780,9.879,400.140,167.044,49.436,159.065
C06778=1022.786,10.128,400.126,167.047,49.432,159.065
C06779=1022.792,10.378,400.113,167.051,49.428,159.065
C06780=1022.798,10.627,400.098,167.053,49.423,159.064
C06781=1022.805,10.911,400.081,167.055,49.418,159.064
C06782=1022.811,11.194,400.065,167.059,49.413,159.063
C06783=1022.818,11.477,400.048,167.062,49.409,159.063
C06784=1022.825,11.761,400.032,167.065,49.404,159.062
C06785=1022.831,12.010,400.017,167.067,49.400,159.062
C06786=1022.837,12.259,400.002,167.071,49.395,159.062
C06787=1022.844,12.509,399.989,167.073,49.391,159.061
C06788=1022.850,12.758,399.974,167.076,49.387,159.061
C06789=1022.856,13.007,399.960,167.079,49.382,159.060
C06790=1022.862,13.258,399.945,167.081,49.378,159.060
C06791=1022.868,13.506,399.931,167.084,49.373,159.060
C06792=1022.874,13.756,399.916,167.086,49.370,159.059
C06793=1022.880,14.005,399.901,167.089,49.366,159.059
C06794=1022.885,14.256,399.887,167.092,49.362,159.059
C06795=1022.891,14.505,399.872,167.094,49.357,159.058
C06796=1022.897,14.754,399.857,167.097,49.353,159.058
C06797=1022.904,15.004,399.842,167.100,49.349,159.057
C06798=1022.909,15.253,399.827,167.102,49.344,159.057
C06799=1022.916,15.503,399.813,167.105,49.340,159.057
C06800=1022.921,15.752,399.798,167.108,49.336,159.056
C06801=1022.927,16.002,399.783,167.110,49.332,159.056
C06802=1022.933,16.251,399.769,167.113,49.328,159.055
C06803=1022.939,16.501,399.754,167.115,49.324,159.055
C06804=1022.945,16.750,399.739,167.118,49.320,159.055
C06805=1022.951,16.999,399.724,167.120,49.315,159.054
C06806=1022.957,17.250,399.709,167.124,49.311,159.054
C06807=1022.962,17.499,399.695,167.127,49.307,159.054
C06808=1022.969,17.749,399.680,167.129,49.302,159.053
C06809=1022.975,17.997,399.665,167.132,49.298,159.053
C06810=1022.981,18.247,399.650,167.135,49.294,159.053
C06811=1022.987,18.497,399.635,167.137,49.289,159.052
C06812=1022.992,18.746,399.620,167.140,49.285,159.052
C06813=1022.999,18.996,399.605,167.143,49.281,159.051
C06814=1023.005,19.245,399.591,167.145,49.277,159.051
C06815=1023.011,19.494,399.576,167.148,49.273,159.051
C06816=1023.017,19.744,399.560,167.150,49.269,159.050
C06817=1023.022,19.993,399.545,167.153,49.264,159.050
C06818=1023.029,20.243,399.531,167.156,49.260,159.049
C06819=1023.034,20.492,399.515,167.158,49.256,159.049
C06820=1023.040,20.742,399.500,167.161,49.251,159.049
C06821=1023.047,20.992,399.485,167.163,49.247,159.048
C06822=1023.052,21.241,399.470,167.166,49.244,159.048
C06823=1023.058,21.490,399.455,167.169,49.240,159.048
C06824=1023.064,21.740,399.440,167.171,49.235,159.047
C06825=1023.069,21.989,399.425,167.174,49.231,159.047
C06826=1023.076,22.239,399.410,167.177,49.227,159.046
C06827=1023.082,22.489,399.395,167.179,49.222,159.046
C06828=1023.087,22.738,399.380,167.182,49.218,159.046
C06829=1023.094,22.988,399.365,167.185,49.214,159.045
C06830=1023.100,23.237,399.350,167.187,49.210,159.045
C06831=1023.105,23.487,399.335,167.190,49.206,159.044
C06832=1023.112,23.736,399.319,167.192,49.201,159.044
C06833=1023.118,23.985,399.304,167.195,49.197,159.044
C06834=1023.123,24.234,399.289,167.198,49.193,159.043
C06835=1023.130,24.484,399.274,167.200,49.188,159.043
C06836=1023.136,24.734,399.259,167.203,49.184,159.042
C06837=1023.141,24.983,399.244,167.206,49.180,159.042
C06838=1023.147,25.233,399.229,167.208,49.176,159.042
C06839=1023.154,25.482,399.214,167.211,49.172,159.041
C06840=1023.159,25.731,399.198,167.213,49.167,159.041
C06841=1023.165,25.981,399.184,167.216,49.163,159.040
C06842=1023.171,26.231,399.168,167.219,49.159,159.040
C06843=1023.177,26.480,399.153,167.221,49.155,159.040
C06844=1023.183,26.729,399.138,167.224,49.151,159.039
C06845=1023.189,27.014,399.121,167.227,49.146,159.039
C06846=1023.197,27.299,399.103,167.229,49.141,159.038
C06847=1023.204,27.584,399.086,167.233,49.136,159.038
C06848=1023.211,27.868,399.068,167.236,49.131,159.038
C06849=1023.216,28.118,399.053,167.239,49.127,159.037
C06850=1023.223,28.367,399.037,167.241,49.122,159.037
C06851=1023.228,28.617,399.022,167.243,49.119,159.036
C06852=1023.234,28.867,399.006,167.246,49.115,159.036
C06853=1023.240,29.115,398.991,167.249,49.111,159.036
C06854=1023.246,29.365,398.975,167.251,49.106,159.035
C06855=1023.252,29.614,398.961,167.254,49.102,159.035
C06856=1023.258,29.864,398.944,167.257,49.098,159.034
C06857=1023.263,30.113,398.929,167.259,49.094,159.034
C06858=1023.270,30.362,398.913,167.262,49.090,159.034
C06859=1023.275,30.612,398.898,167.264,49.086,159.033
C06860=1023.282,30.862,398.883,167.267,49.081,159.033
C06861=1023.288,31.111,398.867,167.270,49.077,159.032
C06862=1023.293,31.360,398.852,167.272,49.073,159.032
C06863=1023.299,31.609,398.836,167.275,49.069,159.032
C06864=1023.305,31.859,398.820,167.277,49.065,159.031
C06865=1023.311,32.109,398.805,167.280,49.061,159.031
C06866=1023.317,32.358,398.789,167.283,49.056,159.030
C06867=1023.323,32.607,398.775,167.285,49.052,159.030
C06868=1023.329,32.857,398.758,167.288,49.047,159.030
C06869=1023.335,33.107,398.743,167.291,49.043,159.029
C06870=1023.341,33.356,398.727,167.293,49.039,159.029
C06871=1023.347,33.606,398.712,167.296,49.035,159.028
C06872=1023.353,33.855,398.697,167.298,49.031,159.028
C06873=1023.359,34.104,398.681,167.301,49.027,159.028
C06874=1023.364,34.354,398.665,167.304,49.022,159.027
C06875=1023.371,34.603,398.650,167.306,49.018,159.027
C06876=1023.377,34.853,398.634,167.309,49.014,159.026
C06877=1023.383,35.102,398.618,167.311,49.010,159.026
C06878=1023.389,35.352,398.603,167.314,49.005,159.026
C06879=1023.394,35.601,398.587,167.317,49.001,159.025
C06880=1023.401,35.850,398.572,167.319,48.997,159.025
C06881=1023.407,36.100,398.556,167.322,48.993,159.024
C06882=1023.413,36.349,398.541,167.325,48.989,159.024
C06883=1023.419,36.599,398.524,167.327,48.984,159.024
C06884=1023.425,36.848,398.508,167.330,48.980,159.023
C06885=1023.431,37.098,398.493,167.332,48.976,159.023
C06886=1023.437,37.347,398.477,167.335,48.971,159.022
C06887=1023.442,37.596,398.462,167.338,48.968,159.022
C06888=1023.448,37.846,398.446,167.340,48.964,159.022
C06889=1023.454,38.095,398.429,167.343,48.959,159.021
C06890=1023.460,38.345,398.414,167.346,48.955,159.021
C06891=1023.466,38.594,398.398,167.348,48.951,159.020
C06892=1023.473,38.843,398.382,167.351,48.946,159.020
C06893=1023.478,39.093,398.366,167.353,48.942,159.020
C06894=1023.484,39.343,398.350,167.356,48.939,159.019
C06895=1023.490,39.592,398.334,167.358,48.934,159.019
C06896=1023.496,39.841,398.318,167.360,48.930,159.018
C06897=1023.501,40.091,398.302,167.363,48.926,159.018
C06898=1023.507,40.340,398.286,167.366,48.922,159.018
C06899=1023.514,40.589,398.270,167.368,48.918,159.017
C06900=1023.519,40.839,398.255,167.371,48.914,159.017
C06901=1023.525,41.088,398.239,167.373,48.909,159.016
C06902=1023.531,41.338,398.222,167.376,48.905,159.016
C06903=1023.537,41.587,398.206,167.379,48.901,159.015
C06904=1023.543,41.837,398.191,167.381,48.897,159.015
C06905=1023.549,42.086,398.174,167.384,48.893,159.015
C06906=1023.556,42.335,398.159,167.387,48.888,159.014
C06907=1023.562,42.585,398.142,167.389,48.884,159.014
C06908=1023.568,42.834,398.126,167.392,48.880,159.014
C06909=1023.574,43.119,398.108,167.395,48.876,159.013
C06910=1023.580,43.403,398.090,167.398,48.871,159.013
C06911=1023.587,43.688,398.071,167.400,48.866,159.012
C06912=1023.594,43.973,398.053,167.404,48.861,159.012
C06913=1023.599,44.222,398.036,167.406,48.858,159.011
C06914=1023.605,44.472,398.020,167.408,48.854,159.011
C06915=1023.611,44.721,398.003,167.411,48.850,159.011
C06916=1023.617,44.970,397.987,167.414,48.845,159.010
C06917=1023.623,45.220,397.971,167.416,48.841,159.010
C06918=1023.629,45.469,397.955,167.419,48.837,159.009
C06919=1023.634,45.718,397.938,167.421,48.833,159.009
C06920=1023.640,45.968,397.922,167.424,48.829,159.009
C06921=1023.646,46.218,397.905,167.427,48.825,159.008
C06922=1023.652,46.467,397.889,167.429,48.821,159.008
C06923=1023.658,46.716,397.873,167.431,48.816,159.007
C06924=1023.663,46.966,397.856,167.434,48.813,159.007
C06925=1023.669,47.215,397.840,167.437,48.809,159.007
C06926=1023.675,47.464,397.824,167.439,48.804,159.006
C06927=1023.681,47.714,397.807,167.442,48.800,159.006
C06928=1023.687,47.963,397.791,167.445,48.796,159.005
C06929=1023.692,48.213,397.775,167.447,48.792,159.005
C06930=1023.698,48.462,397.758,167.450,48.788,159.005
C06931=1023.704,48.711,397.742,167.453,48.784,159.004
C06932=1023.710,48.961,397.726,167.455,48.779,159.004
C06933=1023.716,49.210,397.710,167.457,48.775,159.003
C06934=1023.722,49.460,397.693,167.460,48.771,159.003
C06935=1023.727,49.709,397.676,167.462,48.767,159.002
C06936=1023.733,49.958,397.660,167.465,48.763,159.002
C06937=1023.739,50.208,397.644,167.467,48.759,159.002
C06938=1023.746,50.456,397.627,167.470,48.754,159.001
C06939=1023.752,50.706,397.610,167.473,48.751,159.001
C06940=1023.758,50.956,397.594,167.475,48.747,159.001
C06941=1023.763,51.205,397.577,167.478,48.742,159.000
C06942=1023.769,51.455,397.561,167.481,48.738,159.000
C06943=1023.775,51.704,397.545,167.483,48.733,158.999
C06944=1023.781,51.954,397.528,167.486,48.730,158.999
C06945=1023.787,52.203,397.512,167.489,48.726,158.999
C06946=1023.793,52.452,397.496,167.491,48.721,158.998
C06947=1023.799,52.701,397.478,167.494,48.717,158.998
C06948=1023.805,52.951,397.462,167.495,48.713,158.997
C06949=1023.811,53.200,397.446,167.498,48.709,158.997
C06950=1023.817,53.450,397.429,167.501,48.705,158.996
C06951=1023.823,53.699,397.413,167.503,48.700,158.996
C06952=1023.829,53.949,397.397,167.506,48.696,158.995
C06953=1023.834,54.198,397.379,167.508,48.692,158.995
C06954=1023.840,54.447,397.363,167.511,48.688,158.995
C06955=1023.846,54.696,397.347,167.514,48.683,158.994
C06956=1023.852,54.946,397.330,167.516,48.679,158.994
C06957=1023.859,55.196,397.314,167.519,48.675,158.993
C06958=1023.865,55.445,397.297,167.522,48.671,158.993
C06959=1023.870,55.694,397.280,167.524,48.667,158.993
C06960=1023.876,55.944,397.264,167.527,48.662,158.992
C06961=1023.882,56.193,397.247,167.530,48.658,158.992
C06962=1023.889,56.442,397.230,167.532,48.654,158.991
C06963=1023.895,56.692,397.214,167.535,48.650,158.991
C06964=1023.901,56.941,397.198,167.537,48.645,158.990
C06965=1023.906,57.191,397.181,167.540,48.641,158.990
C06966=1023.912,57.439,397.164,167.542,48.637,158.989
C06967=1023.918,57.689,397.148,167.545,48.633,158.989
C06968=1023.924,57.938,397.131,167.548,48.628,158.989
C06969=1023.931,58.188,397.115,167.550,48.624,158.988
C06970=1023.936,58.437,397.097,167.553,48.620,158.988
C06971=1023.942,58.687,397.081,167.556,48.616,158.987
C06972=1023.948,58.936,397.065,167.558,48.611,158.987
C06973=1023.956,59.220,397.045,167.561,48.607,158.986
C06974=1023.962,59.504,397.026,167.564,48.602,158.986
C06975=1023.969,59.789,397.007,167.566,48.597,158.985
C06976=1023.976,60.074,396.989,167.570,48.592,158.985
C06977=1023.983,60.323,396.971,167.572,48.588,158.984
C06978=1023.989,60.572,396.955,167.575,48.584,158.984
C06979=1023.994,60.822,396.938,167.578,48.579,158.984
C06980=1024.000,61.071,396.921,167.580,48.575,158.983
C06981=1024.007,61.321,396.905,167.583,48.571,158.983
C06982=1024.013,61.570,396.888,167.585,48.566,158.982
C06983=1024.019,61.819,396.871,167.588,48.562,158.982
C06984=1024.025,62.068,396.855,167.591,48.558,158.981
C06985=1024.031,62.318,396.837,167.593,48.554,158.981
C06986=1024.037,62.567,396.821,167.596,48.549,158.980
C06987=1024.043,62.817,396.805,167.598,48.545,158.980
C06988=1024.050,63.066,396.787,167.601,48.541,158.980
C06989=1024.055,63.316,396.770,167.603,48.536,158.979
C06990=1024.061,63.564,396.753,167.606,48.532,158.979
C06991=1024.066,63.814,396.737,167.608,48.529,158.978
C06992=1024.073,64.063,396.719,167.610,48.524,158.978
C06993=1024.079,64.313,396.702,167.613,48.520,158.977
C06994=1024.085,64.562,396.685,167.616,48.516,158.977
C06995=1024.091,64.812,396.668,167.618,48.512,158.977
C06996=1024.097,65.061,396.651,167.621,48.507,158.976
C06997=1024.102,65.310,396.634,167.624,48.503,158.976
C06998=1024.108,65.559,396.617,167.626,48.499,158.975
C06999=1024.114,65.809,396.600,167.629,48.495,158.975
C07000=1024.120,66.058,396.583,167.632,48.491,158.974
C07001=1024.126,66.307,396.566,167.634,48.486,158.974
C07002=1024.133,66.557,396.548,167.637,48.482,158.974
C07003=1024.138,66.807,396.532,167.639,48.478,158.973
C07004=1024.144,67.055,396.515,167.642,48.474,158.973
C07005=1024.150,67.305,396.497,167.644,48.470,158.972
C07006=1024.156,67.554,396.480,167.646,48.466,158.972
C07007=1024.162,67.803,396.463,167.649,48.462,158.971
C07008=1024.169,68.053,396.445,167.652,48.457,158.971
C07009=1024.174,68.303,396.429,167.654,48.453,158.971
C07010=1024.179,68.552,396.411,167.657,48.449,158.970
C07011=1024.186,68.801,396.394,167.660,48.445,158.970
C07012=1024.191,69.051,396.377,167.663,48.441,158.969
C07013=1024.197,69.300,396.359,167.665,48.437,158.969
C07014=1024.204,69.549,396.342,167.668,48.433,158.968
C07015=1024.209,69.798,396.324,167.670,48.428,158.968
C07016=1024.215,70.048,396.308,167.673,48.424,158.968
C07017=1024.221,70.297,396.290,167.676,48.420,158.967
C07018=1024.227,70.546,396.273,167.677,48.416,158.967
C07019=1024.232,70.795,396.255,167.680,48.412,158.966
C07020=1024.239,71.045,396.238,167.682,48.408,158.966
C07021=1024.245,71.294,396.221,167.685,48.404,158.965
C07022=1024.250,71.543,396.203,167.688,48.400,158.965
C07023=1024.256,71.793,396.185,167.691,48.395,158.965
C07024=1024.262,72.042,396.168,167.693,48.391,158.964
C07025=1024.269,72.292,396.150,167.696,48.387,158.964
C07026=1024.274,72.541,396.134,167.699,48.383,158.963
C07027=1024.279,72.790,396.116,167.701,48.378,158.963
C07028=1024.286,73.040,396.099,167.704,48.374,158.962
C07029=1024.292,73.289,396.081,167.707,48.371,158.962
C07030=1024.298,73.539,396.063,167.708,48.366,158.961
C07031=1024.304,73.787,396.046,167.711,48.362,158.961
C07032=1024.310,74.036,396.029,167.713,48.358,158.961
C07033=1024.316,74.286,396.011,167.716,48.354,158.960
C07034=1024.321,74.536,395.994,167.719,48.349,158.960
C07035=1024.328,74.785,395.977,167.721,48.346,158.959
C07036=1024.333,75.034,395.959,167.724,48.342,158.959
C07037=1024.340,75.319,395.939,167.727,48.336,158.958
C07038=1024.347,75.602,395.919,167.730,48.332,158.958
C07039=1024.353,75.887,395.899,167.733,48.327,158.957
C07040=1024.360,76.172,395.879,167.736,48.322,158.957
C07041=1024.366,76.420,395.862,167.739,48.318,158.957
C07042=1024.372,76.670,395.844,167.741,48.314,158.956
C07043=1024.378,76.919,395.826,167.744,48.310,158.956
C07044=1024.384,77.169,395.808,167.747,48.306,158.955
C07045=1024.390,77.418,395.791,167.749,48.301,158.955
C07046=1024.396,77.668,395.773,167.752,48.298,158.954
C07047=1024.401,77.917,395.755,167.753,48.293,158.954
C07048=1024.407,78.166,395.737,167.756,48.289,158.954
C07049=1024.413,78.415,395.719,167.759,48.286,158.953
C07050=1024.419,78.664,395.701,167.761,48.281,158.953
C07051=1024.425,78.914,395.684,167.764,48.277,158.952
C07052=1024.430,79.163,395.666,167.767,48.273,158.952
C07053=1024.437,79.412,395.648,167.770,48.269,158.951
C07054=1024.442,79.661,395.630,167.772,48.265,158.951
C07055=1024.448,79.911,395.613,167.775,48.261,158.951
C07056=1024.454,80.160,395.595,167.777,48.257,158.950
C07057=1024.460,80.409,395.576,167.779,48.253,158.950
C07058=1024.466,80.658,395.559,167.782,48.248,158.949
C07059=1024.472,80.908,395.541,167.785,48.244,158.949
C07060=1024.477,81.157,395.523,167.787,48.241,158.949
C07061=1024.483,81.407,395.505,167.790,48.236,158.948
C07062=1024.489,81.656,395.488,167.793,48.232,158.948
C07063=1024.495,81.905,395.469,167.796,48.228,158.947
C07064=1024.501,82.154,395.452,167.798,48.224,158.947
C07065=1024.507,82.404,395.434,167.801,48.220,158.946
C07066=1024.512,82.653,395.416,167.802,48.216,158.946
C07067=1024.519,82.903,395.398,167.805,48.212,158.945
C07068=1024.524,83.151,395.380,167.808,48.208,158.945
C07069=1024.531,83.401,395.362,167.810,48.203,158.945
C07070=1024.536,83.650,395.344,167.813,48.200,158.944
C07071=1024.542,83.900,395.326,167.816,48.195,158.944
C07072=1024.548,84.148,395.308,167.818,48.191,158.943
C07073=1024.554,84.398,395.290,167.821,48.187,158.943
C07074=1024.560,84.647,395.272,167.824,48.183,158.942
C07075=1024.566,84.896,395.255,167.827,48.179,158.942
C07076=1024.572,85.146,395.236,167.829,48.174,158.942
C07077=1024.578,85.395,395.218,167.832,48.171,158.941
C07078=1024.584,85.644,395.201,167.834,48.166,158.941
C07079=1024.589,85.893,395.183,167.837,48.162,158.940
C07080=1024.595,86.143,395.164,167.840,48.158,158.940
C07081=1024.601,86.393,395.146,167.841,48.154,158.939
C07082=1024.607,86.642,395.128,167.844,48.149,158.939
C07083=1024.613,86.891,395.110,167.847,48.146,158.938
C07084=1024.619,87.140,395.092,167.849,48.141,158.938
C07085=1024.625,87.390,395.074,167.852,48.137,158.938
C07086=1024.631,87.639,395.055,167.855,48.133,158.937
C07087=1024.637,87.888,395.038,167.857,48.129,158.937
C07088=1024.643,88.137,395.020,167.860,48.125,158.936
C07089=1024.649,88.386,395.002,167.863,48.120,158.936
C07090=1024.655,88.636,394.984,167.865,48.117,158.935
C07091=1024.661,88.885,394.966,167.868,48.112,158.935
C07092=1024.667,89.134,394.948,167.871,48.108,158.935
C07093=1024.673,89.384,394.930,167.873,48.104,158.934
C07094=1024.679,89.633,394.911,167.876,48.100,158.934
C07095=1024.684,89.882,394.893,167.879,48.095,158.933
C07096=1024.690,90.131,394.874,167.881,48.091,158.933
C07097=1024.696,90.381,394.856,167.884,48.088,158.932
C07098=1024.702,90.630,394.837,167.887,48.083,158.932
C07099=1024.708,90.879,394.819,167.888,48.080,158.931
C07100=1024.713,91.128,394.800,167.891,48.076,158.931
C07101=1024.720,91.413,394.780,167.895,48.071,158.931
C07102=1024.727,91.697,394.759,167.897,48.066,158.930
C07103=1024.733,91.981,394.738,167.901,48.062,158.930
C07104=1024.740,92.265,394.717,167.903,48.057,158.929
C07105=1024.746,92.515,394.699,167.906,48.053,158.929
C07106=1024.752,92.764,394.680,167.909,48.049,158.928
C07107=1024.757,93.013,394.662,167.911,48.045,158.928
C07108=1024.763,93.262,394.643,167.914,48.040,158.927
C07109=1024.769,93.512,394.624,167.917,48.036,158.927
C07110=1024.775,93.761,394.606,167.920,48.033,158.927
C07111=1024.781,94.010,394.588,167.922,48.028,158.926
C07112=1024.786,94.260,394.569,167.925,48.024,158.926
C07113=1024.792,94.508,394.551,167.926,48.020,158.925
C07114=1024.799,94.757,394.532,167.929,48.016,158.925
C07115=1024.804,95.007,394.514,167.932,48.012,158.924
C07116=1024.810,95.256,394.495,167.934,48.008,158.924
C07117=1024.816,95.505,394.477,167.937,48.004,158.924
C07118=1024.822,95.755,394.458,167.940,48.000,158.923
C07119=1024.828,96.003,394.440,167.943,47.996,158.923
C07120=1024.834,96.253,394.421,167.945,47.992,158.922
C07121=1024.839,96.503,394.403,167.948,47.987,158.922
C07122=1024.846,96.752,394.384,167.951,47.983,158.921
C07123=1024.851,97.000,394.365,167.953,47.979,158.921
C07124=1024.857,97.250,394.347,167.956,47.975,158.921
C07125=1024.863,97.499,394.329,167.959,47.971,158.920
C07126=1024.869,97.749,394.309,167.961,47.967,158.920
C07127=1024.875,97.998,394.292,167.964,47.963,158.919
C07128=1024.881,98.247,394.273,167.967,47.958,158.919
C07129=1024.887,98.496,394.254,167.970,47.955,158.918
C07130=1024.893,98.745,394.235,167.972,47.950,158.918
C07131=1024.899,98.995,394.218,167.975,47.946,158.918
C07132=1024.904,99.244,394.199,167.977,47.942,158.917
C07133=1024.911,99.493,394.180,167.980,47.938,158.917
C07134=1024.917,99.743,394.161,167.983,47.933,158.916
C07135=1024.923,99.992,394.142,167.986,47.930,158.916
C07136=1024.928,100.241,394.124,167.987,47.926,158.915
C07137=1024.933,100.490,394.105,167.990,47.922,158.915
C07138=1024.940,100.740,394.086,167.993,47.918,158.914
C07139=1024.946,100.989,394.067,167.996,47.914,158.914
C07140=1024.951,101.238,394.048,167.998,47.910,158.914
C07141=1024.957,101.487,394.029,168.001,47.906,158.913
C07142=1024.963,101.736,394.010,168.004,47.902,158.913
C07143=1024.968,101.986,393.991,168.007,47.898,158.912
C07144=1024.975,102.235,393.972,168.009,47.893,158.912
C07145=1024.980,102.484,393.953,168.012,47.890,158.912
C07146=1024.986,102.733,393.934,168.015,47.886,158.911
C07147=1024.992,102.983,393.916,168.017,47.881,158.911
C07148=1024.997,103.232,393.897,168.020,47.877,158.910
C07149=1025.003,103.482,393.877,168.023,47.874,158.910
C07150=1025.009,103.730,393.859,168.024,47.869,158.909
C07151=1025.015,103.979,393.840,168.027,47.866,158.909
C07152=1025.021,104.229,393.821,168.030,47.862,158.909
C07153=1025.027,104.478,393.802,168.033,47.857,158.908
C07154=1025.032,104.727,393.783,168.035,47.853,158.908
C07155=1025.038,104.976,393.765,168.038,47.849,158.907
C07156=1025.044,105.225,393.745,168.041,47.845,158.907
C07157=1025.050,105.475,393.726,168.044,47.841,158.906
C07158=1025.056,105.724,393.707,168.046,47.837,158.906
C07159=1025.062,105.973,393.688,168.049,47.833,158.906
C07160=1025.067,106.223,393.669,168.052,47.829,158.905
C07161=1025.074,106.471,393.650,168.054,47.825,158.905
C07162=1025.079,106.720,393.631,168.057,47.821,158.904
C07163=1025.085,106.969,393.611,168.060,47.816,158.904
C07164=1025.091,107.218,393.593,168.062,47.813,158.903
C07165=1025.098,107.503,393.571,168.065,47.808,158.903
C07166=1025.104,107.788,393.549,168.068,47.803,158.902
C07167=1025.111,108.072,393.528,168.072,47.799,158.902
C07168=1025.118,108.355,393.506,168.075,47.794,158.901
C07169=1025.124,108.605,393.487,168.077,47.790,158.901
C07170=1025.129,108.854,393.467,168.080,47.786,158.901
C07171=1025.136,109.103,393.449,168.083,47.782,158.900
C07172=1025.141,109.353,393.429,168.085,47.777,158.900
C07173=1025.147,109.602,393.410,168.088,47.774,158.899
C07174=1025.154,109.851,393.392,168.091,47.770,158.899
C07175=1025.160,110.100,393.372,168.093,47.765,158.898
C07176=1025.165,110.350,393.352,168.096,47.762,158.898
C07177=1025.171,110.599,393.333,168.099,47.758,158.898
C07178=1025.177,110.848,393.314,168.102,47.753,158.897
C07179=1025.183,111.097,393.294,168.104,47.749,158.897
C07180=1025.189,111.346,393.275,168.107,47.746,158.896
C07181=1025.194,111.595,393.256,168.110,47.741,158.896
C07182=1025.200,111.845,393.237,168.113,47.737,158.895
C07183=1025.206,112.093,393.217,168.115,47.734,158.895
C07184=1025.212,112.343,393.198,168.118,47.729,158.895
C07185=1025.217,112.592,393.179,168.121,47.725,158.894
C07186=1025.223,112.842,393.159,168.124,47.721,158.894
C07187=1025.229,113.090,393.140,168.126,47.717,158.893
C07188=1025.235,113.340,393.120,168.129,47.713,158.893
C07189=1025.241,113.589,393.100,168.132,47.709,158.893
C07190=1025.246,113.838,393.081,168.134,47.706,158.892
C07191=1025.252,114.088,393.062,168.137,47.702,158.892
C07192=1025.257,114.337,393.041,168.139,47.698,158.891
C07193=1025.263,114.586,393.022,168.142,47.694,158.891
C07194=1025.269,114.835,393.002,168.145,47.690,158.890
C07195=1025.275,115.084,392.983,168.148,47.686,158.890
C07196=1025.281,115.333,392.963,168.150,47.682,158.890
C07197=1025.286,115.583,392.944,168.153,47.678,158.889
C07198=1025.292,115.832,392.924,168.156,47.674,158.889
C07199=1025.297,116.081,392.904,168.159,47.670,158.889
C07200=1025.303,116.331,392.885,168.162,47.667,158.888
C07201=1025.308,116.579,392.865,168.164,47.662,158.888
C07202=1025.314,116.828,392.846,168.167,47.658,158.887
C07203=1025.320,117.077,392.826,168.170,47.654,158.887
C07204=1025.326,117.326,392.807,168.173,47.651,158.887
C07205=1025.332,117.575,392.787,168.175,47.647,158.886
C07206=1025.337,117.825,392.767,168.178,47.642,158.886
C07207=1025.343,118.074,392.747,168.181,47.639,158.885
C07208=1025.349,118.323,392.727,168.184,47.635,158.885
C07209=1025.355,118.573,392.707,168.186,47.631,158.885
C07210=1025.361,118.822,392.687,168.189,47.627,158.884
C07211=1025.367,119.071,392.668,168.192,47.623,158.884
C07212=1025.373,119.320,392.648,168.195,47.619,158.883
C07213=1025.377,119.570,392.628,168.198,47.615,158.883
C07214=1025.383,119.818,392.608,168.199,47.611,158.882
C07215=1025.389,120.067,392.588,168.202,47.607,158.882
C07216=1025.395,120.317,392.569,168.205,47.603,158.882
C07217=1025.401,120.565,392.549,168.207,47.599,158.881
C07218=1025.407,120.815,392.530,168.210,47.595,158.881
C07219=1025.413,121.064,392.510,168.213,47.591,158.880
C07220=1025.418,121.313,392.489,168.217,47.587,158.880
C07221=1025.424,121.562,392.470,168.219,47.583,158.879
C07222=1025.430,121.811,392.450,168.222,47.579,158.879
C07223=1025.435,122.060,392.431,168.225,47.575,158.879
C07224=1025.441,122.309,392.411,168.228,47.572,158.878
C07225=1025.447,122.558,392.391,168.230,47.567,158.878
C07226=1025.453,122.809,392.371,168.233,47.563,158.877
C07227=1025.459,123.057,392.351,168.236,47.559,158.877
C07228=1025.465,123.306,392.331,168.239,47.555,158.876
C07229=1025.472,123.590,392.309,168.241,47.551,158.876
C07230=1025.479,123.874,392.286,168.245,47.547,158.876
C07231=1025.484,124.158,392.263,168.248,47.542,158.875
C07232=1025.492,124.443,392.240,168.251,47.537,158.875
C07233=1025.497,124.692,392.221,168.254,47.533,158.874
C07234=1025.503,124.941,392.201,168.257,47.529,158.874
C07235=1025.509,125.190,392.180,168.259,47.525,158.873
C07236=1025.515,125.439,392.160,168.262,47.521,158.873
C07237=1025.521,125.689,392.141,168.265,47.517,158.872
C07238=1025.527,125.938,392.121,168.268,47.513,158.872
C07239=1025.533,126.186,392.101,168.272,47.509,158.872
C07240=1025.539,126.435,392.081,168.274,47.505,158.871
C07241=1025.547,126.773,392.054,168.277,47.499,158.871
C07242=1025.554,127.111,392.027,168.282,47.494,158.870
C07243=1025.562,127.449,392.000,168.285,47.489,158.870
C07244=1025.570,127.787,391.973,168.290,47.483,158.869
C07245=1025.576,128.036,391.953,168.292,47.479,158.869
C07246=1025.582,128.285,391.933,168.295,47.475,158.868
C07247=1025.588,128.534,391.913,168.298,47.471,158.868
C07248=1025.594,128.782,391.893,168.300,47.467,158.867
C07249=1025.600,129.032,391.872,168.303,47.463,158.867
C07250=1025.606,129.282,391.853,168.306,47.459,158.866
C07251=1025.612,129.531,391.833,168.309,47.455,158.866
C07252=1025.618,129.779,391.813,168.311,47.451,158.866
C07253=1025.624,130.028,391.793,168.315,47.447,158.865
C07254=1025.631,130.278,391.772,168.318,47.443,158.865
C07255=1025.636,130.527,391.752,168.321,47.439,158.864
C07256=1025.641,130.776,391.731,168.324,47.435,158.864
C07257=1025.647,131.025,391.711,168.326,47.431,158.864
C07258=1025.653,131.275,391.690,168.329,47.428,158.863
C07259=1025.659,131.523,391.670,168.332,47.423,158.863
C07260=1025.664,131.773,391.650,168.335,47.419,158.862
C07261=1025.670,132.021,391.630,168.338,47.416,158.862
C07262=1025.675,132.270,391.609,168.340,47.412,158.862
C07263=1025.682,132.520,391.589,168.343,47.408,158.861
C07264=1025.687,132.769,391.568,168.346,47.404,158.861
C07265=1025.693,133.018,391.549,168.349,47.400,158.860
C07266=1025.699,133.267,391.528,168.352,47.396,158.860
C07267=1025.705,133.517,391.508,168.354,47.392,158.860
C07268=1025.711,133.765,391.486,168.357,47.389,158.859
C07269=1025.717,134.014,391.466,168.360,47.385,158.859
C07270=1025.722,134.263,391.446,168.364,47.380,158.858
C07271=1025.729,134.512,391.426,168.367,47.376,158.858
C07272=1025.734,134.762,391.405,168.370,47.373,158.858
C07273=1025.740,135.010,391.385,168.372,47.369,158.857
C07274=1025.746,135.260,391.364,168.375,47.365,158.857
C07275=1025.752,135.509,391.344,168.378,47.361,158.856
C07276=1025.757,135.758,391.323,168.381,47.357,158.856
C07277=1025.762,136.007,391.302,168.384,47.353,158.856
C07278=1025.769,136.256,391.282,168.386,47.349,158.855
C07279=1025.774,136.505,391.261,168.389,47.346,158.855
C07280=1025.780,136.754,391.241,168.392,47.341,158.854
C07281=1025.786,137.003,391.220,168.395,47.337,158.854
C07282=1025.792,137.252,391.199,168.399,47.333,158.854
C07283=1025.798,137.501,391.179,168.401,47.330,158.853
